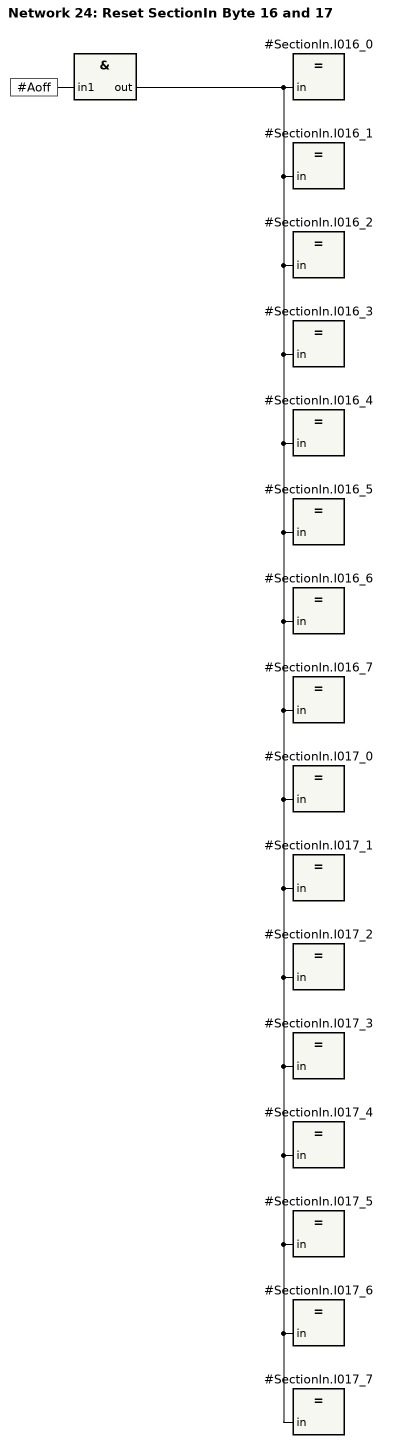
   #SectionIn.I016_0 := #Aoff;
   #SectionIn.I016_1 := #Aoff;
   #SectionIn.I016_2 := #Aoff;
   #SectionIn.I016_3 := #Aoff;
   #SectionIn.I016_4 := #Aoff;
   #SectionIn.I016_5 := #Aoff;
   #SectionIn.I016_6 := #Aoff;
   #SectionIn.I016_7 := #Aoff;
   #SectionIn.I017_0 := #Aoff;
   #SectionIn.I017_1 := #Aoff;
   #SectionIn.I017_2 := #Aoff;
   #SectionIn.I017_3 := #Aoff;
   #SectionIn.I017_4 := #Aoff;
   #SectionIn.I017_5 := #Aoff;
   #SectionIn.I017_6 := #Aoff;
   #SectionIn.I017_7 := #Aoff;
END_REGION

REGION Network 25: Reset SectionIn Byte 18 and 19
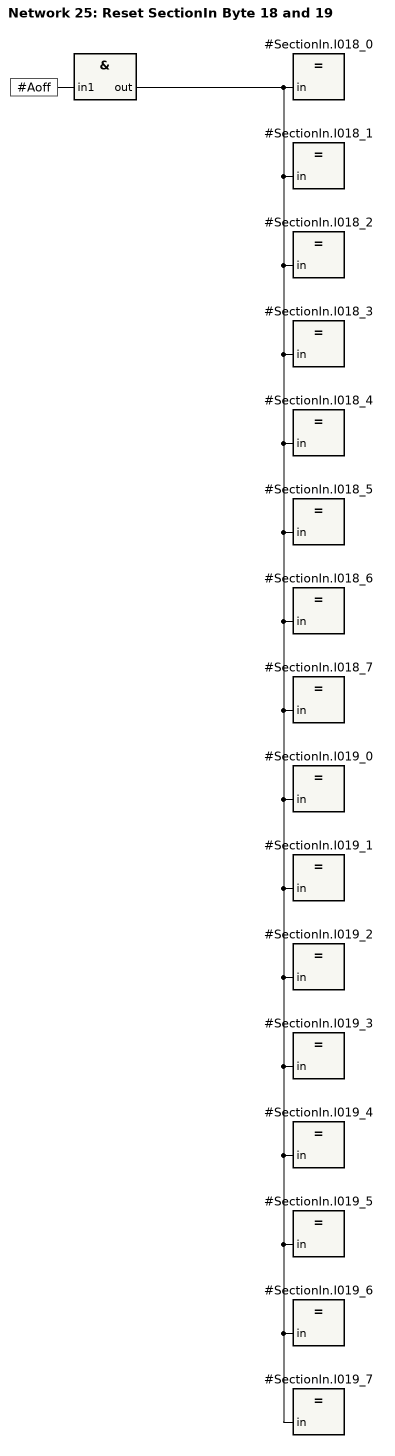
   #SectionIn.I018_0 := #Aoff;
   #SectionIn.I018_1 := #Aoff;
   #SectionIn.I018_2 := #Aoff;
   #SectionIn.I018_3 := #Aoff;
   #SectionIn.I018_4 := #Aoff;
   #SectionIn.I018_5 := #Aoff;
   #SectionIn.I018_6 := #Aoff;
   #SectionIn.I018_7 := #Aoff;
   #SectionIn.I019_0 := #Aoff;
   #SectionIn.I019_1 := #Aoff;
   #SectionIn.I019_2 := #Aoff;
   #SectionIn.I019_3 := #Aoff;
   #SectionIn.I019_4 := #Aoff;
   #SectionIn.I019_5 := #Aoff;
   #SectionIn.I019_6 := #Aoff;
   #SectionIn.I019_7 := #Aoff;
END_REGION

REGION Network 26: Reset SectionIn Byte 20 and 21
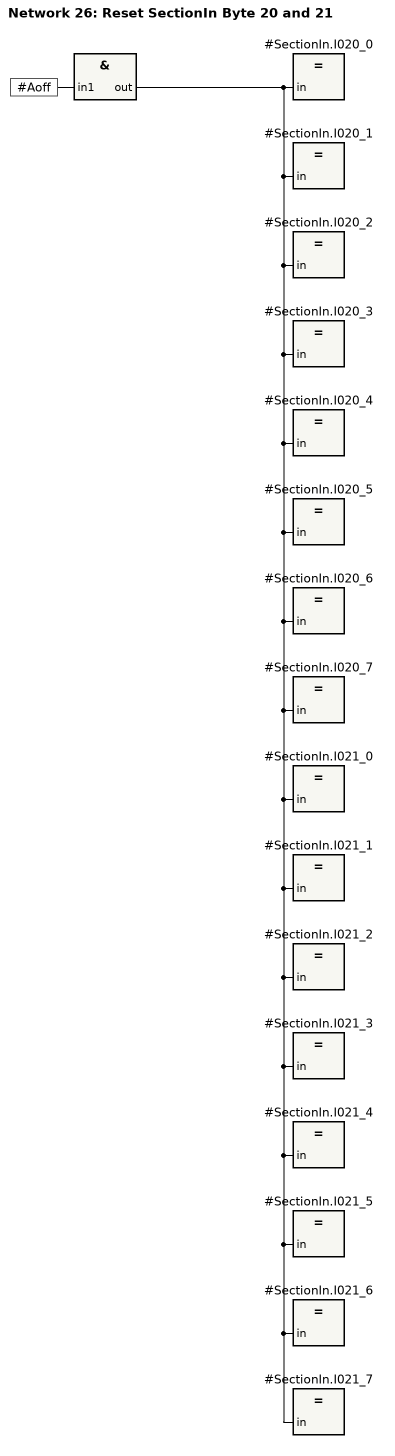
   #SectionIn.I020_0 := #Aoff;
   #SectionIn.I020_1 := #Aoff;
   #SectionIn.I020_2 := #Aoff;
   #SectionIn.I020_3 := #Aoff;
   #SectionIn.I020_4 := #Aoff;
   #SectionIn.I020_5 := #Aoff;
   #SectionIn.I020_6 := #Aoff;
   #SectionIn.I020_7 := #Aoff;
   #SectionIn.I021_0 := #Aoff;
   #SectionIn.I021_1 := #Aoff;
   #SectionIn.I021_2 := #Aoff;
   #SectionIn.I021_3 := #Aoff;
   #SectionIn.I021_4 := #Aoff;
   #SectionIn.I021_5 := #Aoff;
   #SectionIn.I021_6 := #Aoff;
   #SectionIn.I021_7 := #Aoff;
END_REGION

REGION Network 27: Reset SectionIn 22 to 99
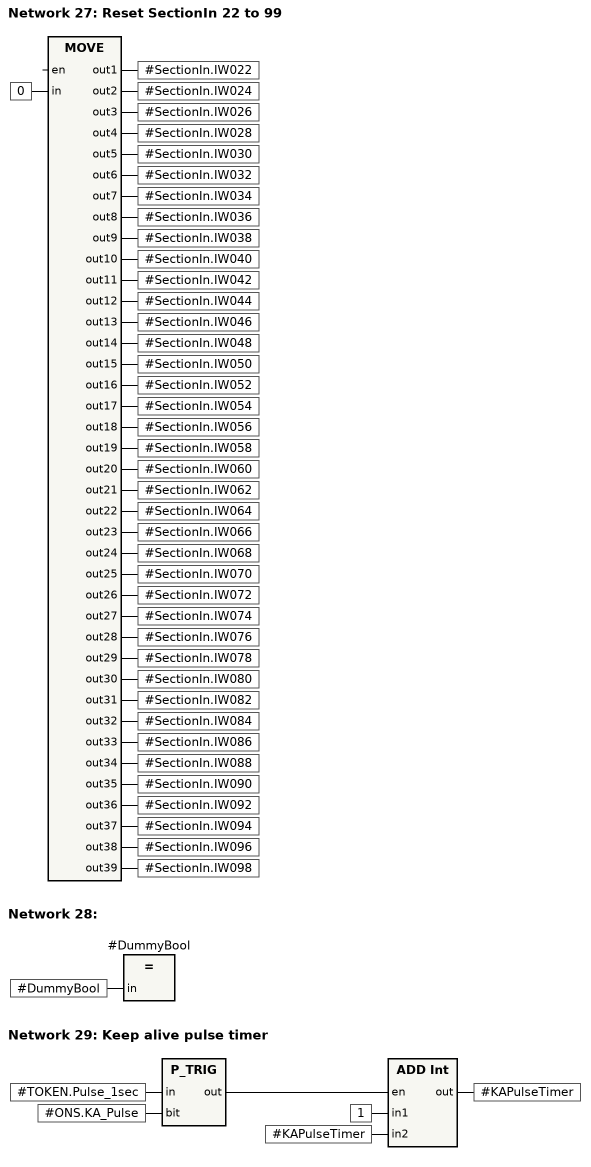
   #SectionIn.IW022 := 0;
   #SectionIn.IW024 := 0;
   #SectionIn.IW026 := 0;
   #SectionIn.IW028 := 0;
   #SectionIn.IW030 := 0;
   #SectionIn.IW032 := 0;
   #SectionIn.IW034 := 0;
   #SectionIn.IW036 := 0;
   #SectionIn.IW038 := 0;
   #SectionIn.IW040 := 0;
   #SectionIn.IW042 := 0;
   #SectionIn.IW044 := 0;
   #SectionIn.IW046 := 0;
   #SectionIn.IW048 := 0;
   #SectionIn.IW050 := 0;
   #SectionIn.IW052 := 0;
   #SectionIn.IW054 := 0;
   #SectionIn.IW056 := 0;
   #SectionIn.IW058 := 0;
   #SectionIn.IW060 := 0;
   #SectionIn.IW062 := 0;
   #SectionIn.IW064 := 0;
   #SectionIn.IW066 := 0;
   #SectionIn.IW068 := 0;
   #SectionIn.IW070 := 0;
   #SectionIn.IW072 := 0;
   #SectionIn.IW074 := 0;
   #SectionIn.IW076 := 0;
   #SectionIn.IW078 := 0;
   #SectionIn.IW080 := 0;
   #SectionIn.IW082 := 0;
   #SectionIn.IW084 := 0;
   #SectionIn.IW086 := 0;
   #SectionIn.IW088 := 0;
   #SectionIn.IW090 := 0;
   #SectionIn.IW092 := 0;
   #SectionIn.IW094 := 0;
   #SectionIn.IW096 := 0;
   #SectionIn.IW098 := 0;
END_REGION

REGION Network 28
   Res1:
   #DummyBool := #DummyBool;
END_REGION

REGION Network 29: Keep alive pulse timer
   #_w1 := #TOKEN.Pulse_1sec AND NOT #ONS.KA_Pulse;   // rising edge
   #ONS.KA_Pulse := #TOKEN.Pulse_1sec;
   IF #_w1 THEN #KAPulseTimer := 1 + #KAPulseTimer; END_IF;
END_REGION

REGION Network 30: Keep alive pulse generated
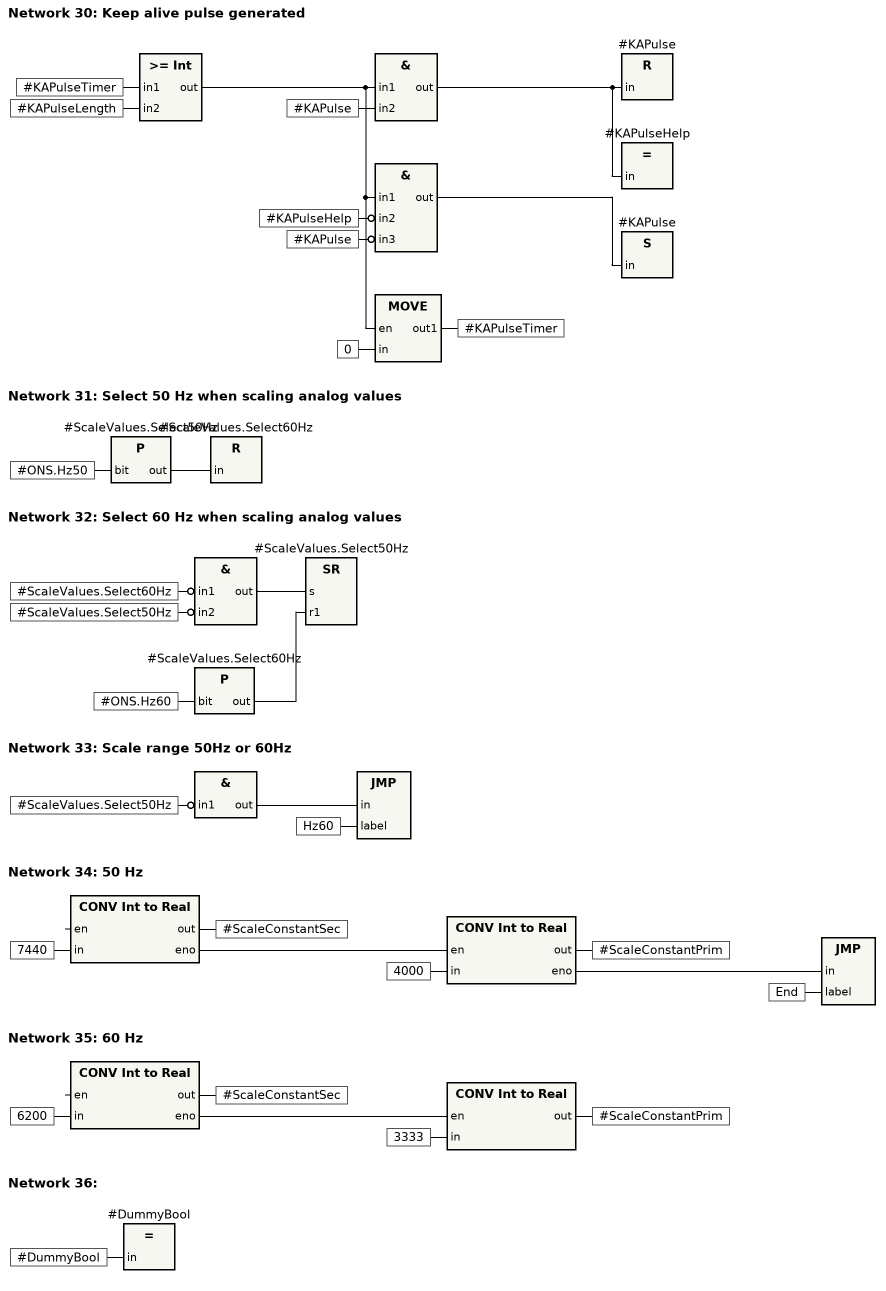
   #_w1 := #KAPulseTimer >= #KAPulseLength;
   #_w2 := #_w1 AND #KAPulse;
   IF #_w2 THEN #KAPulse := FALSE; END_IF;
   #KAPulseHelp := #_w2;
   IF #_w1 AND NOT #KAPulseHelp AND NOT #KAPulse THEN #KAPulse := TRUE; END_IF;
   IF #_w1 THEN #KAPulseTimer := 0; END_IF;
END_REGION

REGION Network 31: Select 50 Hz when scaling analog values
   #_w1 := #ScaleValues.Select50Hz AND NOT #ONS.Hz50;   // rising edge of #ScaleValues.Select50Hz
   #ONS.Hz50 := #ScaleValues.Select50Hz;
   IF #_w1 THEN #ScaleValues.Select60Hz := FALSE; END_IF;
END_REGION

REGION Network 32: Select 60 Hz when scaling analog values
   #_w1 := #ScaleValues.Select60Hz AND NOT #ONS.Hz60;   // rising edge of #ScaleValues.Select60Hz
   #ONS.Hz60 := #ScaleValues.Select60Hz;
   IF NOT #ScaleValues.Select60Hz AND NOT #ScaleValues.Select50Hz THEN
       #ScaleValues.Select50Hz := TRUE;   // SR flip-flop
   END_IF;
   IF #_w1 THEN #ScaleValues.Select50Hz := FALSE; END_IF;
END_REGION

REGION Network 33: Scale range 50Hz or 60Hz
   // Jump if not 50Hz
   IF NOT #ScaleValues.Select50Hz THEN GOTO Hz60; END_IF;
END_REGION

REGION Network 34: 50 Hz
   #ScaleConstantSec := INT_TO_REAL(7440);
   #ScaleConstantPrim := INT_TO_REAL(4000);
   GOTO End;
END_REGION

REGION Network 35: 60 Hz
   Hz60:
   #ScaleConstantSec := INT_TO_REAL(6200);
   #ScaleConstantPrim := INT_TO_REAL(3333);
END_REGION

REGION Network 36
   End:
   #DummyBool := #DummyBool;
END_REGION

REGION Network 37: Latch Acknowledge signal from ECS section
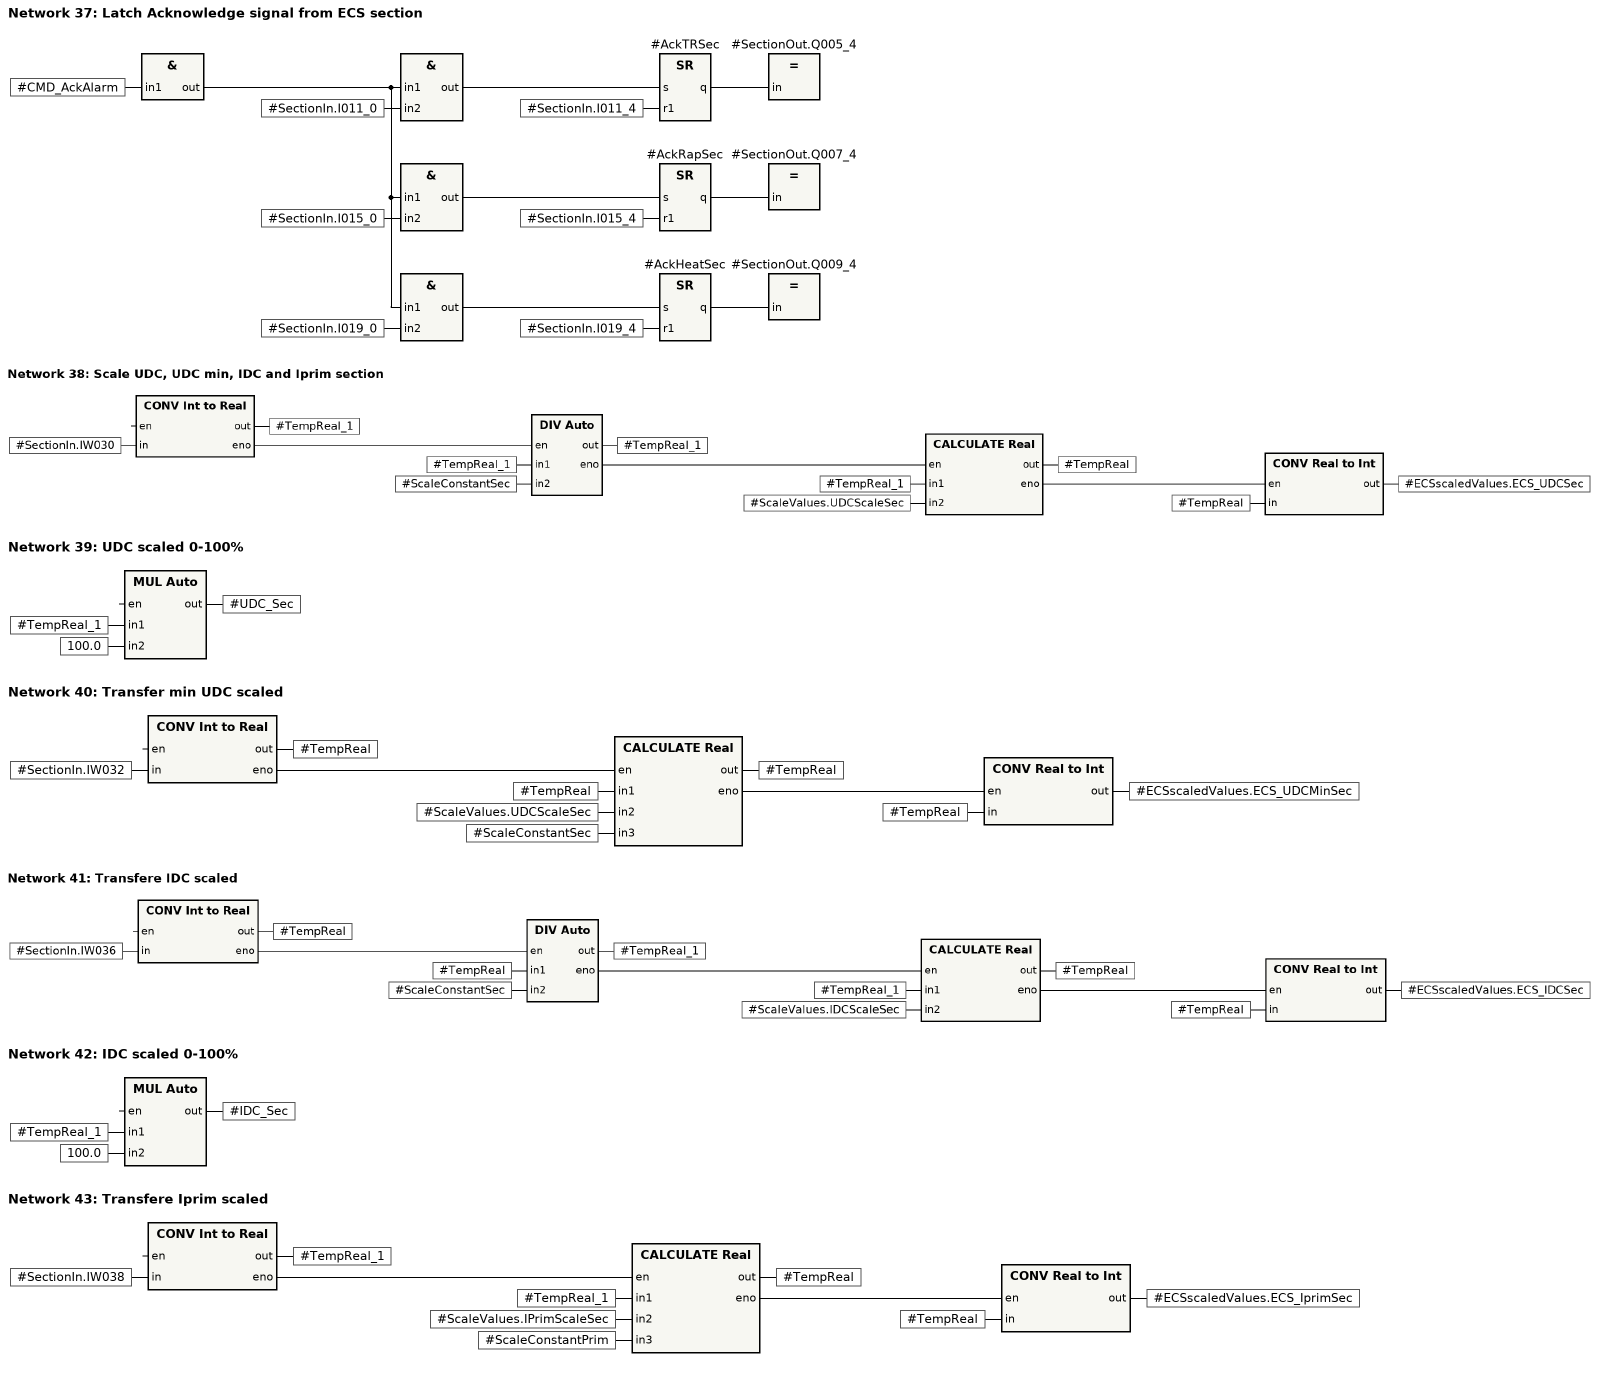
   IF #CMD_AckAlarm AND #SectionIn.I011_0 THEN
       #AckTRSec := TRUE;   // SR flip-flop
   END_IF;
   IF #SectionIn.I011_4 THEN #AckTRSec := FALSE; END_IF;
   #SectionOut.Q005_4 := #AckTRSec;
   IF #CMD_AckAlarm AND #SectionIn.I015_0 THEN
       #AckRapSec := TRUE;   // SR flip-flop
   END_IF;
   IF #SectionIn.I015_4 THEN #AckRapSec := FALSE; END_IF;
   #SectionOut.Q007_4 := #AckRapSec;
   IF #CMD_AckAlarm AND #SectionIn.I019_0 THEN
       #AckHeatSec := TRUE;   // SR flip-flop
   END_IF;
   IF #SectionIn.I019_4 THEN #AckHeatSec := FALSE; END_IF;
   #SectionOut.Q009_4 := #AckHeatSec;
END_REGION

REGION Network 38: Scale UDC, UDC min, IDC and Iprim section
   // Transfer UDC scaled
   // Build 002 : 26 March 2019 - ECS_UDCSec/ECS_UDCMinSec were mul by 10.0 before and the same is removed
   #TempReal_1 := INT_TO_REAL(#SectionIn.IW030);
   #TempReal_1 := #TempReal_1 / #ScaleConstantSec;
   #TempReal := ROUND(#TempReal_1*#ScaleValues.UDCScaleSec);
   #ECSscaledValues.ECS_UDCSec := REAL_TO_INT(#TempReal);
END_REGION

REGION Network 39: UDC scaled 0-100%
   #UDC_Sec := #TempReal_1 * 100.0;
END_REGION

REGION Network 40: Transfer min UDC scaled
   // Build 002 : 26 March 2019 - ECS_UDCSec/ECS_UDCMinSec were mul by 10.0 before and the same is removed
   #TempReal := INT_TO_REAL(#SectionIn.IW032);
   #TempReal := ROUND((#TempReal*#ScaleValues.UDCScaleSec)/#ScaleConstantSec);
   #ECSscaledValues.ECS_UDCMinSec := REAL_TO_INT(#TempReal);
END_REGION

REGION Network 41: Transfere IDC scaled
   #TempReal := INT_TO_REAL(#SectionIn.IW036);
   #TempReal_1 := #TempReal / #ScaleConstantSec;
   #TempReal := ROUND(#TempReal_1*#ScaleValues.IDCScaleSec);
   #ECSscaledValues.ECS_IDCSec := REAL_TO_INT(#TempReal);
END_REGION

REGION Network 42: IDC scaled 0-100%
   #IDC_Sec := #TempReal_1 * 100.0;
END_REGION

REGION Network 43: Transfere Iprim scaled
   #TempReal_1 := INT_TO_REAL(#SectionIn.IW038);
   #TempReal := ROUND((#TempReal_1*#ScaleValues.IPrimScaleSec)/#ScaleConstantPrim);
   #ECSscaledValues.ECS_IprimSec := REAL_TO_INT(#TempReal);
END_REGION

REGION Network 44: Transfer general outputs to gateway
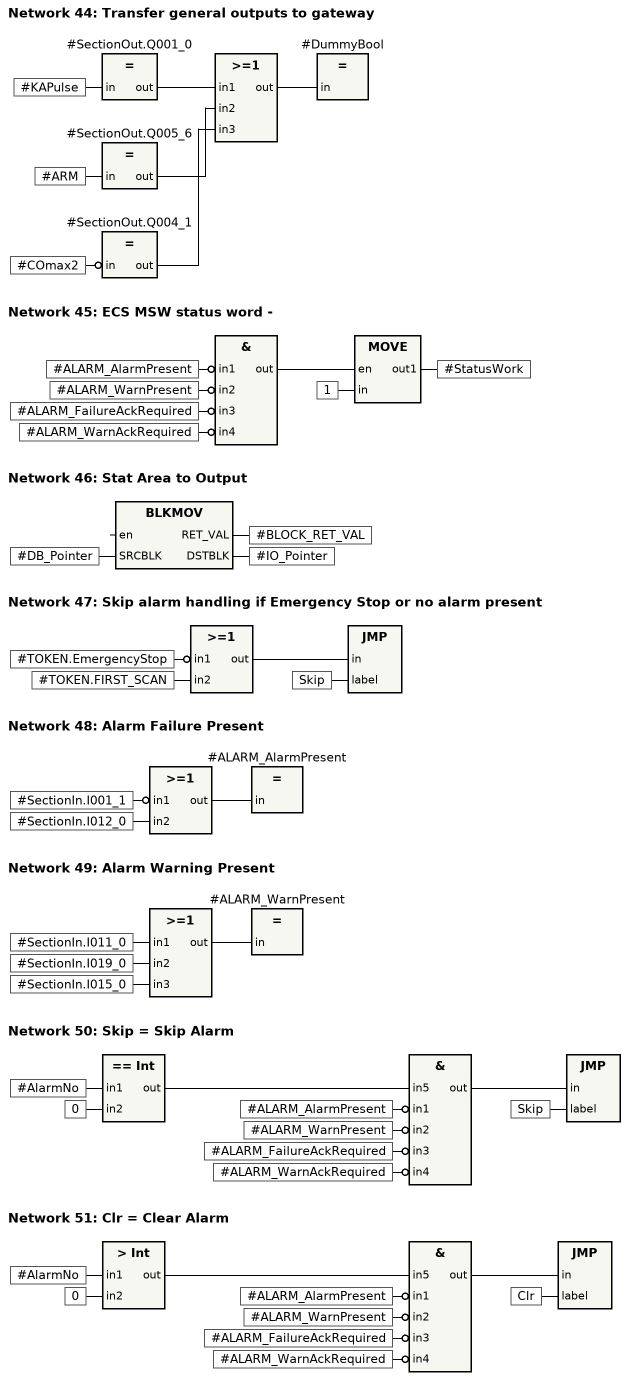
   #SectionOut.Q001_0 := #KAPulse;
   #SectionOut.Q005_6 := #ARM;
   #SectionOut.Q004_1 := NOT #COmax2;
   #DummyBool := #KAPulse OR #ARM OR NOT #COmax2;
END_REGION

REGION Network 45: ECS MSW status word -
   IF NOT #ALARM_AlarmPresent AND NOT #ALARM_WarnPresent AND NOT #ALARM_FailureAckRequired AND NOT #ALARM_WarnAckRequired THEN
       #StatusWork := 1;
   END_IF;
END_REGION

REGION Network 46: Stat Area to Output
   #BLOCK_RET_VAL := BLKMOV(SRCBLK := #DB_Pointer, DSTBLK => #IO_Pointer);
END_REGION

REGION Network 47: Skip alarm handling if Emergency Stop or no alarm present
   // Skip = Skip Alarm
   IF NOT #TOKEN.EmergencyStop OR #TOKEN.FIRST_SCAN THEN GOTO Skip; END_IF;
END_REGION

REGION Network 48: Alarm Failure Present
   #ALARM_AlarmPresent := NOT #SectionIn.I001_1 OR #SectionIn.I012_0;
END_REGION

REGION Network 49: Alarm Warning Present
   #ALARM_WarnPresent := #SectionIn.I011_0 OR #SectionIn.I019_0 OR #SectionIn.I015_0;
END_REGION

REGION Network 50: Skip = Skip Alarm
   IF (#AlarmNo = 0) AND NOT #ALARM_AlarmPresent AND NOT #ALARM_WarnPresent AND NOT #ALARM_FailureAckRequired AND NOT #ALARM_WarnAckRequired THEN
       GOTO Skip;
   END_IF;
END_REGION

REGION Network 51: Clr = Clear Alarm
   IF (#AlarmNo > 0) AND NOT #ALARM_AlarmPresent AND NOT #ALARM_WarnPresent AND NOT #ALARM_FailureAckRequired AND NOT #ALARM_WarnAckRequired THEN
       GOTO Clr;
   END_IF;
END_REGION

REGION Network 52: Ack = Alarm Acknowledge
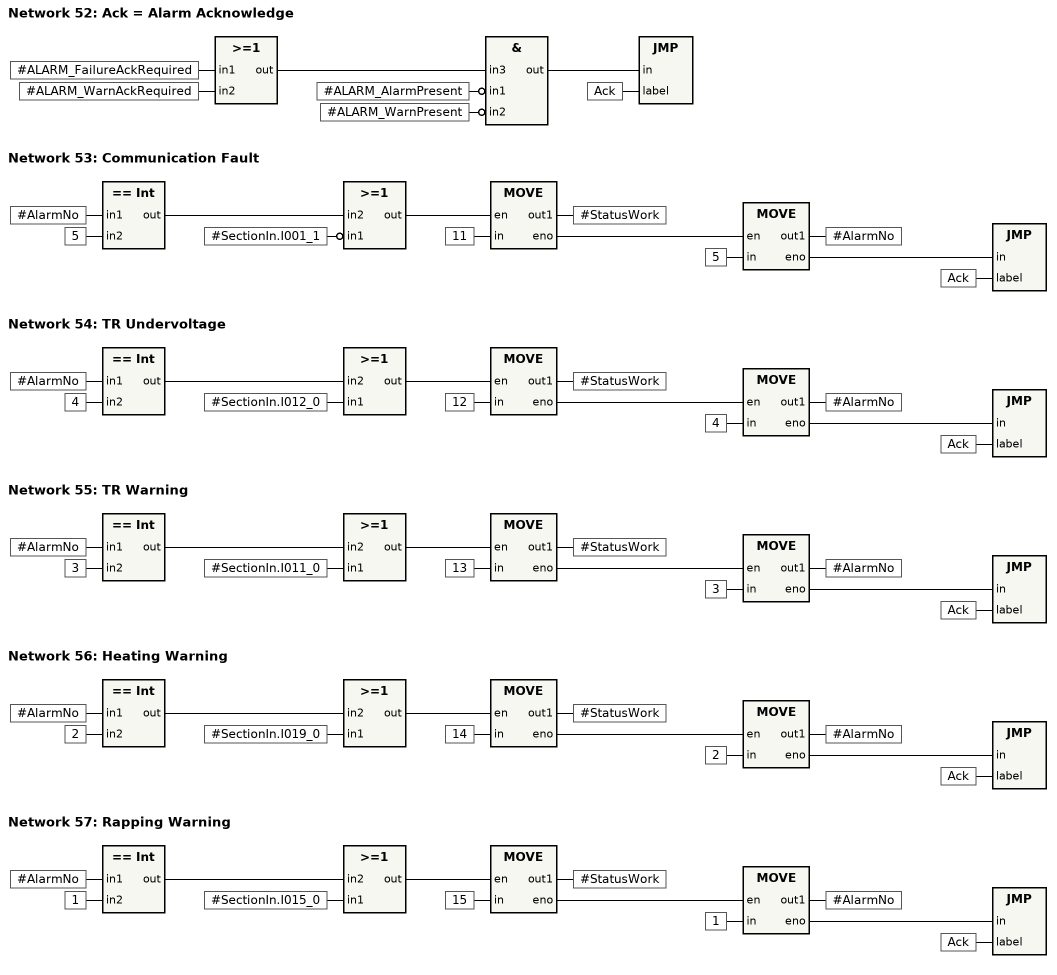
   IF (#ALARM_FailureAckRequired OR #ALARM_WarnAckRequired) AND NOT #ALARM_AlarmPresent AND NOT #ALARM_WarnPresent THEN
       GOTO Ack;
   END_IF;
END_REGION

REGION Network 53: Communication Fault
   // ENO of a box is taken as its EN; it also drops when the box reports an error
   #_w1 := (#AlarmNo = 5) OR NOT #SectionIn.I001_1;
   IF #_w1 THEN
       #StatusWork := 11;
       #AlarmNo := 5;
       GOTO Ack;
   END_IF;
END_REGION

REGION Network 54: TR Undervoltage
   // ENO of a box is taken as its EN; it also drops when the box reports an error
   #_w1 := (#AlarmNo = 4) OR #SectionIn.I012_0;
   IF #_w1 THEN
       #StatusWork := 12;
       #AlarmNo := 4;
       GOTO Ack;
   END_IF;
END_REGION

REGION Network 55: TR Warning
   // ENO of a box is taken as its EN; it also drops when the box reports an error
   #_w1 := (#AlarmNo = 3) OR #SectionIn.I011_0;
   IF #_w1 THEN
       #StatusWork := 13;
       #AlarmNo := 3;
       GOTO Ack;
   END_IF;
END_REGION

REGION Network 56: Heating Warning
   // ENO of a box is taken as its EN; it also drops when the box reports an error
   #_w1 := (#AlarmNo = 2) OR #SectionIn.I019_0;
   IF #_w1 THEN
       #StatusWork := 14;
       #AlarmNo := 2;
       GOTO Ack;
   END_IF;
END_REGION

REGION Network 57: Rapping Warning
   // ENO of a box is taken as its EN; it also drops when the box reports an error
   #_w1 := (#AlarmNo = 1) OR #SectionIn.I015_0;
   IF #_w1 THEN
       #StatusWork := 15;
       #AlarmNo := 1;
       GOTO Ack;
   END_IF;
END_REGION

REGION Network 58: Alarm Acknowledge
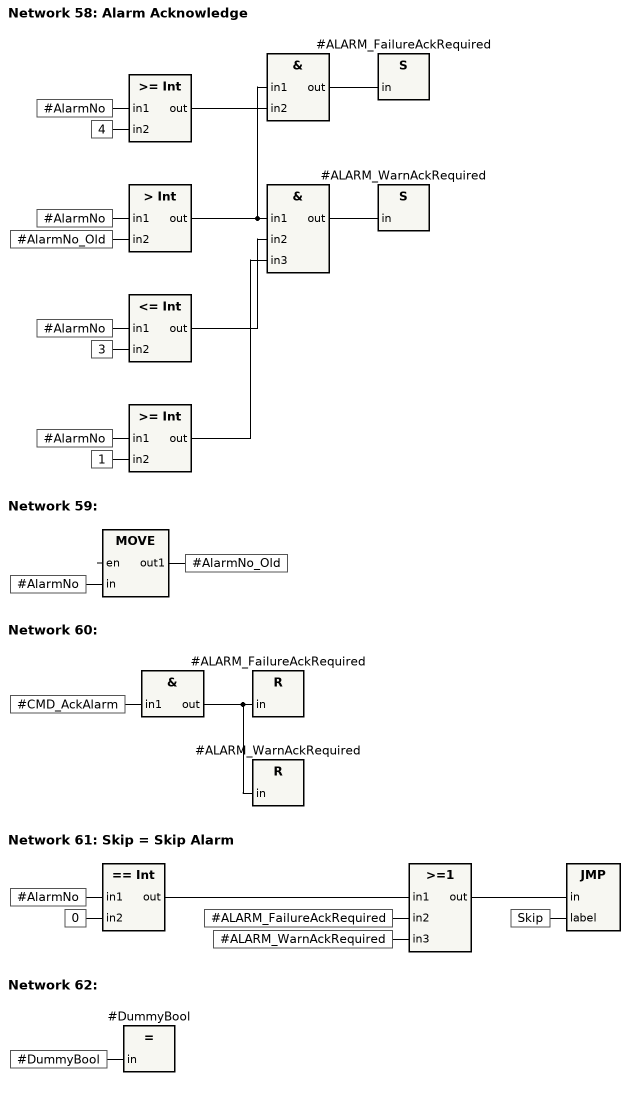
   Ack:
   #_w1 := #AlarmNo > #AlarmNo_Old;
   IF #_w1 AND (#AlarmNo >= 4) THEN #ALARM_FailureAckRequired := TRUE; END_IF;
   IF #_w1 AND (#AlarmNo <= 3) AND (#AlarmNo >= 1) THEN #ALARM_WarnAckRequired := TRUE; END_IF;
END_REGION

REGION Network 59
   #AlarmNo_Old := #AlarmNo;
END_REGION

REGION Network 60
   IF #CMD_AckAlarm THEN
       #ALARM_FailureAckRequired := FALSE;
       #ALARM_WarnAckRequired := FALSE;
   END_IF;
END_REGION

REGION Network 61: Skip = Skip Alarm
   IF (#AlarmNo = 0) OR #ALARM_FailureAckRequired OR #ALARM_WarnAckRequired THEN GOTO Skip; END_IF;
END_REGION

REGION Network 62
   Clr:
   #DummyBool := #DummyBool;
END_REGION

REGION Network 63
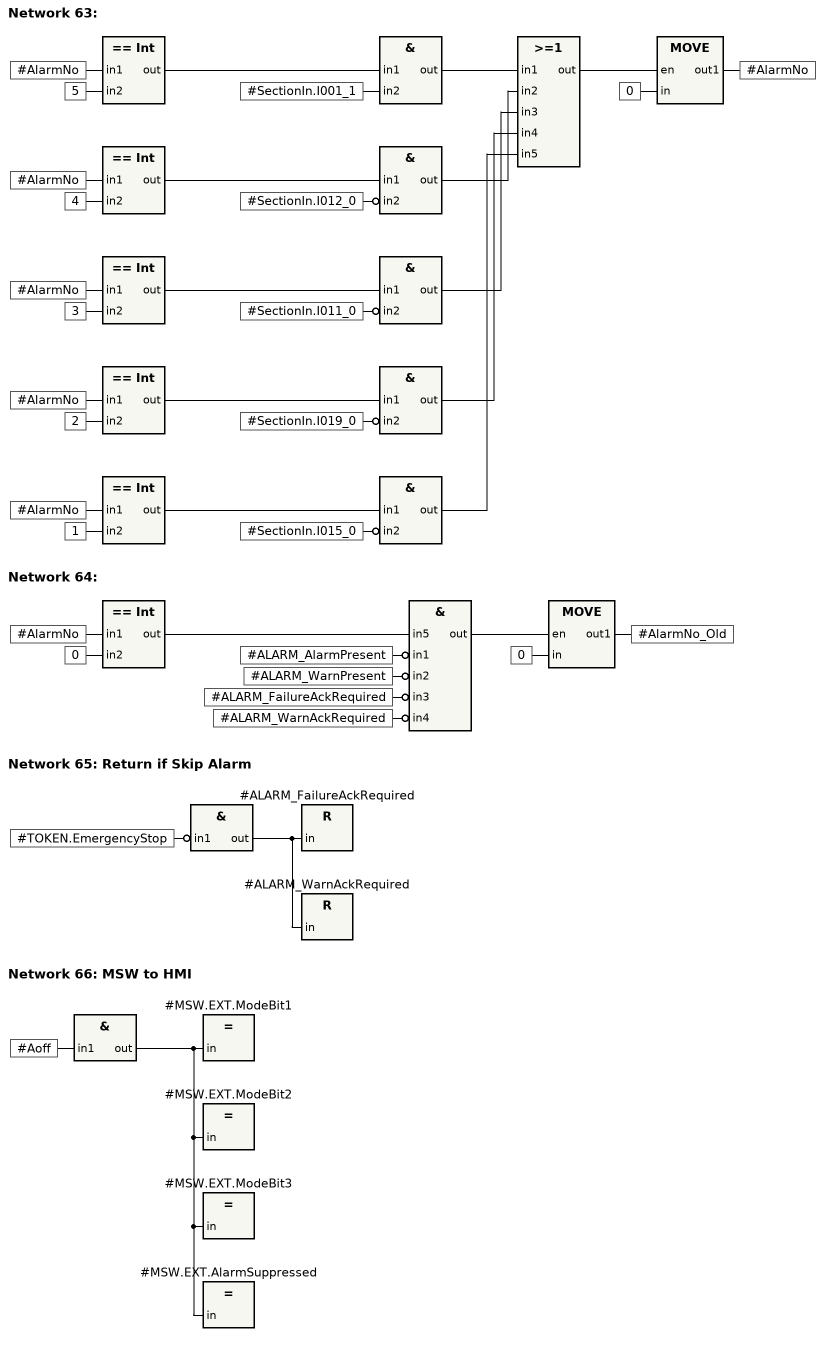
   IF ((#AlarmNo = 5) AND #SectionIn.I001_1) OR ((#AlarmNo = 4) AND NOT #SectionIn.I012_0) OR ((#AlarmNo = 3) AND NOT #SectionIn.I011_0) OR ((#AlarmNo = 2) AND NOT #SectionIn.I019_0) OR ((#AlarmNo = 1) AND NOT #SectionIn.I015_0) THEN
       #AlarmNo := 0;
   END_IF;
END_REGION

REGION Network 64
   IF (#AlarmNo = 0) AND NOT #ALARM_AlarmPresent AND NOT #ALARM_WarnPresent AND NOT #ALARM_FailureAckRequired AND NOT #ALARM_WarnAckRequired THEN
       #AlarmNo_Old := 0;
   END_IF;
END_REGION

REGION Network 65: Return if Skip Alarm
   Skip:
   IF NOT #TOKEN.EmergencyStop THEN
       #ALARM_FailureAckRequired := FALSE;
       #ALARM_WarnAckRequired := FALSE;
   END_IF;
END_REGION

REGION Network 66: MSW to HMI
   #MSW.EXT.ModeBit1 := #Aoff;
   #MSW.EXT.ModeBit2 := #Aoff;
   #MSW.EXT.ModeBit3 := #Aoff;
   #MSW.EXT.AlarmSuppressed := #Aoff;
END_REGION

REGION Network 67
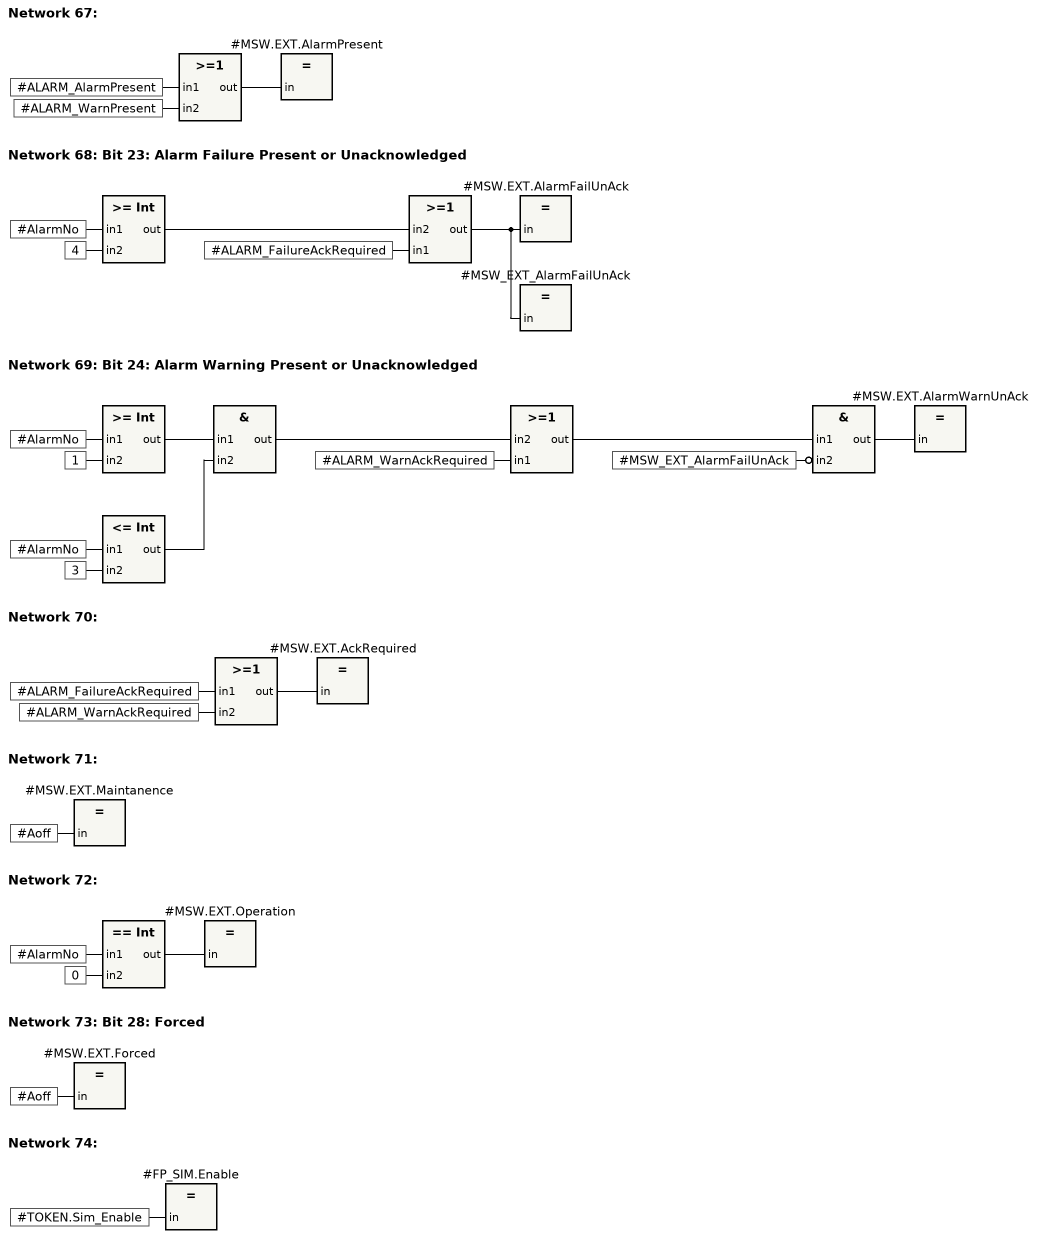
   #MSW.EXT.AlarmPresent := #ALARM_AlarmPresent OR #ALARM_WarnPresent;
END_REGION

REGION Network 68: Bit 23: Alarm Failure Present or Unacknowledged
   #MSW.EXT.AlarmFailUnAck := (#AlarmNo >= 4) OR #ALARM_FailureAckRequired;
   #MSW_EXT_AlarmFailUnAck := #MSW.EXT.AlarmFailUnAck;
END_REGION

REGION Network 69: Bit 24: Alarm Warning Present or Unacknowledged
   #MSW.EXT.AlarmWarnUnAck := (((#AlarmNo >= 1) AND (#AlarmNo <= 3)) OR #ALARM_WarnAckRequired) AND NOT #MSW_EXT_AlarmFailUnAck;
END_REGION

REGION Network 70
   #MSW.EXT.AckRequired := #ALARM_FailureAckRequired OR #ALARM_WarnAckRequired;
END_REGION

REGION Network 71
   #MSW.EXT.Maintanence := #Aoff;
END_REGION

REGION Network 72
   #MSW.EXT.Operation := #AlarmNo = 0;
END_REGION

REGION Network 73: Bit 28: Forced
   #MSW.EXT.Forced := #Aoff;
END_REGION

REGION Network 74
   #FP_SIM.Enable := #TOKEN.Sim_Enable;
END_REGION

REGION Network 75: MSW & TIMESTAMP TO HMI
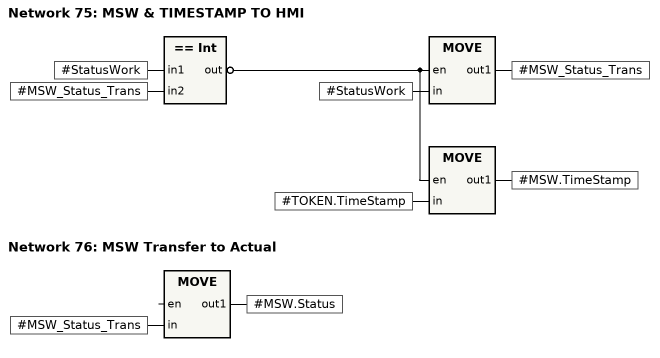
   #_w1 := NOT (#StatusWork = #MSW_Status_Trans);
   IF #_w1 THEN
       #MSW_Status_Trans := #StatusWork;
       #MSW.TimeStamp := #TOKEN.TimeStamp;
   END_IF;
END_REGION

REGION Network 76: MSW Transfer to Actual
   #MSW.Status := #MSW_Status_Trans;
END_REGION
END_FUNCTION_BLOCK

FUNCTION_BLOCK "ACESYS_SEL_ANALOG"   // FB234, FBD
TITLE = ACESYS V8.0 - Build 002 - Select Analog Block
{ S7_Optimized_Access := 'FALSE' }
AUTHOR : FLSmidth
FAMILY : ACESYS
NAME : SEL_ALOG
VERSION : 8.0
   VAR_INPUT
      X1 : Real;   // Signal 1
      X2 : Real;   // Signal 2
      X3 : Real;   // Signal 3
      X1_OK : Bool;   // Signal 1 Enable
      X2_OK : Bool;   // Signal 2 Enable
      X3_OK : Bool;   // Signal 3 Enable
   END_VAR
   VAR_OUTPUT
      SEL_X1 : Bool;   // Signal 1 Selected
      SEL_X2 : Bool;   // Signal 2 Selected
      SEL_X3 : Bool;   // Signal 3 Selected
      AL_X1 : Bool;   // Alarm Signal 1 (1 = OK)
      AL_X2 : Bool;   // Alarm Signal 2 (1 = OK)
      AL_X3 : Bool;   // Alarm Signal 3 (1 = OK)
      AVG : Real;   // Average
      MSW : "ACESYS_HMI_STAT_ANALOG";
   END_VAR
   VAR_IN_OUT
      TOKEN : "ACESYS_TOKEN";
   END_VAR
   VAR
      BlockInfo : Struct
         Ace_Version : Int;   // Acesys Block Version Number
         Ace_BuildNo : Int;   // Acesys Block Build Number
         DB_Number : Int;   // Block Instance DB Number
      END_STRUCT;
      FP_CMD : Struct   // Faceplate Commands
         Spare_08 : Bool;
         Spare_09 : Bool;
         Spare_10 : Bool;
         Spare_11 : Bool;
         Spare_12 : Bool;
         Spare_13 : Bool;
         Spare_14 : Bool;
         AckAlarm : Bool;
         Spare_00 : Bool;
         Spare_01 : Bool;
         Spare_02 : Bool;
         Spare_03 : Bool;
         Spare_04 : Bool;
         Spare_05 : Bool;
         Spare_06 : Bool;
         Spare_07 : Bool;
      END_STRUCT;
      FP_SEL : Struct   // Faceplate Selection
         X1 : Bool := TRUE;   // Select X1 from Faceplate
         X2 : Bool := TRUE;   // Select X2 from Faceplate
         X3 : Bool := TRUE;   // Select X3 from Faceplate
         Type2 : Bool;   // Select 2 Sensors
         Type3 : Bool;   // Select 3 Sensors
         MaxVal : Bool;   // Select Max Value (2 sensors)
         MinVal : Bool;   // Select Min Value (2 sensors)
         Spare9 : Bool;
         Spare8 : Bool;
         Spare7 : Bool;
         Spare6 : Bool;
         Spare5 : Bool;
         Spare4 : Bool;
         Spare3 : Bool;
         Spare2 : Bool;
         Spare1 : Bool;
      END_STRUCT;
      FP_SHOW : Struct   // Faceplate Show Object
         X1 : Bool;   // Show X1 on Faceplate
         X2 : Bool;   // Show X2 on Faceplate
         X3 : Bool;   // Show X3 on Faceplate
      END_STRUCT;
      FP_PARM : Struct   // Faceplate Parameters
         MaxDiff : Real := 10.0;   // Max Diff SP
         AL_Delay_Pre : Int := 3;   // Alarm Delay Pre
         AL_Delay_Acc : Int;   // Alarm Delay ACC
      END_STRUCT;
      ONS : Struct
         SecPulse1 : Bool;   // Oneshot Bit
         SecPulse2 : Bool;   // Oneshot Bit
         Sel_Type2 : Bool;   // Oneshot Bit
         Sel_Type3 : Bool;   // Oneshot Bit
         Sel_High : Bool;   // Oneshot Bit
         Sel_Low : Bool;   // Oneshot Bit
         Sel_Max : Bool;   // Oneshot Bit
         Sel_Min : Bool;   // Oneshot Bit
         Acknowledge : Bool;
         Spare7 : Bool;
         Spare6 : Bool;
         Spare5 : Bool;
         Spare4 : Bool;
         Spare3 : Bool;
         Spare2 : Bool;
         Spare1 : Bool;
      END_STRUCT;
      Sec_Pulse : Bool;   // Pulse Every Second
      Sig1_3_NotOK : Bool;
      Sig1_2_NotOK : Bool;
      Sig2_3_NotOK : Bool;
      Sig1_Deviation : Bool;   // Signal 1 Deviation
      Sig2_Deviation : Bool;   // Signal 2 Deviation
      Sig3_Deviation : Bool;   // Signal 3 Deviation
      CMD_Acknowledge : Bool;   // Internal Acknowledge
      ALARM_SuppresionActiv : Bool;   // Internal Alarm Supression
      ALARM_AlarmPresent : Bool;
      ALARM_Failure_Ack_Requ : Bool;
      ALARM_Warn_Ack_Requ : Bool;
      ALARM_WarnPresent : Bool;
      SEL_X1_int : Bool;   // Signal 1 Selected
      SEL_X2_int : Bool;   // Signal 2 Selected
      SEL_X3_int : Bool;   // Signal 3 Selected
      Sig1_Fault : Bool;   // Signal 1 Fault
      Sig2_Fault : Bool;   // Signal 2 Fault
      Sig3_Fault : Bool;   // Signal 3 Fault
      Sig1_3_TimerMEM : Int;   // Timer Memory Register
      Sig1_2_TimerMEM : Int;   // Timer Memory Register
      Sig2_3_TimerMEM : Int;   // Timer Memory Register
      AlarmNo : Int;   // Alarm Number
      AlarmNo_Old : Int;   // Old Alarm Number
      StatusWork : Int;   // Internal ECS Status
      No_X : Real;   // Number of Signals in Calculation
      Sum_X : Real;   // Total Signal Value of X:s
      MinMaxVal : Real;   // Selected Min Max Val (for Type-2)
      OUT : Struct
         SEL_X1 : Bool;
         SEL_X2 : Bool;
         SEL_X3 : Bool;
         AL_X1 : Bool;
         AL_X2 : Bool;
         AL_X3 : Bool;
         AVG : Real;
         MSW_EXT_ALARMFAILUNACK : Bool;
      END_STRUCT;
      MSW_Status_Trans : Int;
   END_VAR
   VAR_TEMP
      AOn : Bool;   // Always On
      AOff : Bool;   // Always Off
      DummyBool : Bool;
      DummyReal_1 : Real;
      DummyReal_2 : Real;
   END_VAR
   VAR_TEMP   // added for the SCL form of the ladder/FBD networks
      _w1 : Bool;
      _w2 : Bool;
   END_VAR
BEGIN

REGION Network 1: Always On
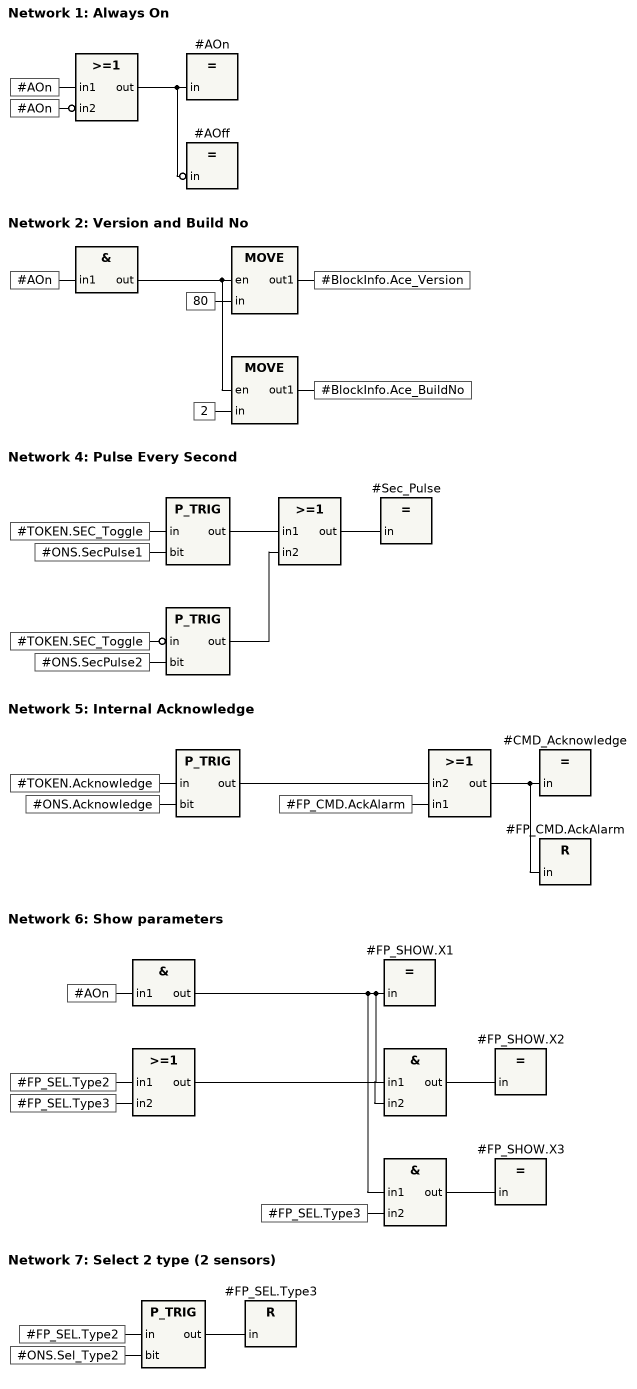
   #AOn := #AOn OR NOT #AOn;
   #AOff := NOT #AOn;
END_REGION

REGION Network 2: Version and Build No
   IF #AOn THEN
       #BlockInfo.Ace_Version := 80;
       #BlockInfo.Ace_BuildNo := 2;
   END_IF;
END_REGION

REGION Network 3 (STL): Instance DB Number to Faceplate
         L     DINO;
         T     #BlockInfo.DB_Number;
END_REGION

REGION Network 4: Pulse Every Second
   #_w1 := #TOKEN.SEC_Toggle AND NOT #ONS.SecPulse1;   // rising edge
   #ONS.SecPulse1 := #TOKEN.SEC_Toggle;
   #_w2 := NOT #TOKEN.SEC_Toggle AND NOT #ONS.SecPulse2;   // rising edge
   #ONS.SecPulse2 := NOT #TOKEN.SEC_Toggle;
   #Sec_Pulse := #_w1 OR #_w2;
END_REGION

REGION Network 5: Internal Acknowledge
   #_w1 := #TOKEN.Acknowledge AND NOT #ONS.Acknowledge;   // rising edge
   #ONS.Acknowledge := #TOKEN.Acknowledge;
   #CMD_Acknowledge := #_w1 OR #FP_CMD.AckAlarm;
   IF #CMD_Acknowledge THEN #FP_CMD.AckAlarm := FALSE; END_IF;
END_REGION

REGION Network 6: Show parameters
   #FP_SHOW.X1 := #AOn;
   #FP_SHOW.X2 := #AOn AND (#FP_SEL.Type2 OR #FP_SEL.Type3);
   #FP_SHOW.X3 := #AOn AND #FP_SEL.Type3;
END_REGION

REGION Network 7: Select 2 type (2 sensors)
   #_w1 := #FP_SEL.Type2 AND NOT #ONS.Sel_Type2;   // rising edge
   #ONS.Sel_Type2 := #FP_SEL.Type2;
   IF #_w1 THEN #FP_SEL.Type3 := FALSE; END_IF;
END_REGION

REGION Network 8: Select 3 type (3 sensors)
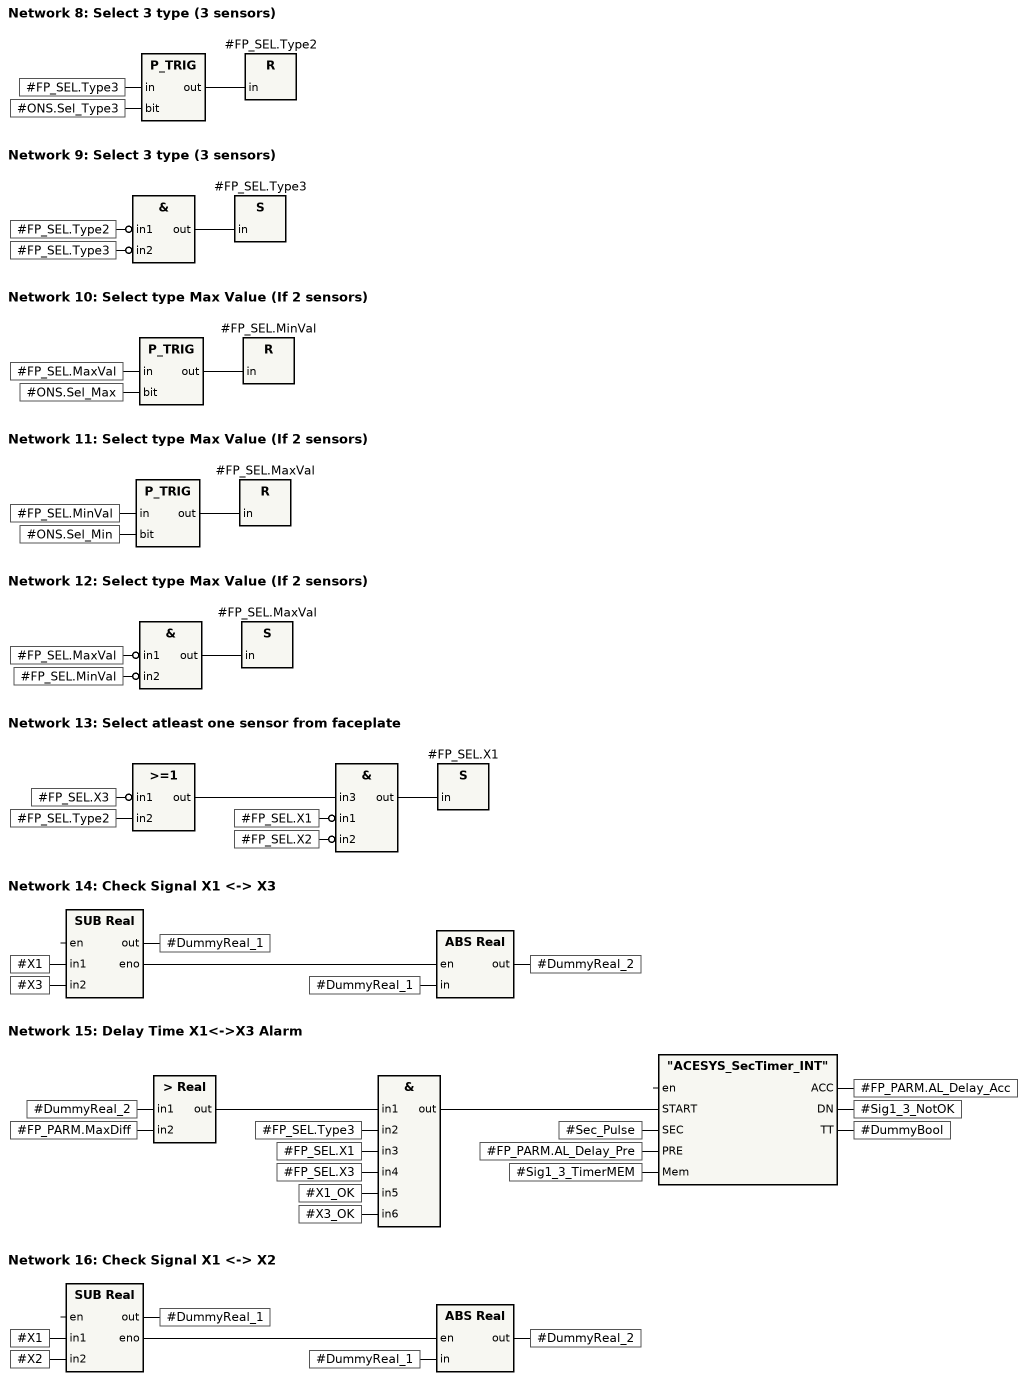
   #_w1 := #FP_SEL.Type3 AND NOT #ONS.Sel_Type3;   // rising edge
   #ONS.Sel_Type3 := #FP_SEL.Type3;
   IF #_w1 THEN #FP_SEL.Type2 := FALSE; END_IF;
END_REGION

REGION Network 9: Select 3 type (3 sensors)
   IF NOT #FP_SEL.Type2 AND NOT #FP_SEL.Type3 THEN #FP_SEL.Type3 := TRUE; END_IF;
END_REGION

REGION Network 10: Select type Max Value (If 2 sensors)
   #_w1 := #FP_SEL.MaxVal AND NOT #ONS.Sel_Max;   // rising edge
   #ONS.Sel_Max := #FP_SEL.MaxVal;
   IF #_w1 THEN #FP_SEL.MinVal := FALSE; END_IF;
END_REGION

REGION Network 11: Select type Max Value (If 2 sensors)
   #_w1 := #FP_SEL.MinVal AND NOT #ONS.Sel_Min;   // rising edge
   #ONS.Sel_Min := #FP_SEL.MinVal;
   IF #_w1 THEN #FP_SEL.MaxVal := FALSE; END_IF;
END_REGION

REGION Network 12: Select type Max Value (If 2 sensors)
   IF NOT #FP_SEL.MaxVal AND NOT #FP_SEL.MinVal THEN #FP_SEL.MaxVal := TRUE; END_IF;
END_REGION

REGION Network 13: Select atleast one sensor from faceplate
   // Build 002 - 17. Jun 2019 (EXTBOB) : Faceplate selection for configuration of 
   // analog signal atleast one selected newly added
   IF (NOT #FP_SEL.X3 OR #FP_SEL.Type2) AND NOT #FP_SEL.X1 AND NOT #FP_SEL.X2 THEN
       #FP_SEL.X1 := TRUE;
   END_IF;
END_REGION

REGION Network 14: Check Signal X1 <-> X3
   // ENO of a box is taken as its EN; it also drops when the box reports an error
   #DummyReal_1 := #X1 - #X3;
   #DummyReal_2 := ABS(#DummyReal_1);
END_REGION

REGION Network 15: Delay Time X1<->X3 Alarm
   // Ignor if type-2 Sensor Selecetd
   // 
   // Build 002 - 17. Jun 2019 (EXTBOB) : Faceplate selection & Signal enable 
   // flag added
   "ACESYS_SecTimer_INT"(START := (#DummyReal_2 > #FP_PARM.MaxDiff) AND #FP_SEL.Type3 AND #FP_SEL.X1 AND #FP_SEL.X3 AND #X1_OK AND #X3_OK,
                         SEC := #Sec_Pulse,
                         PRE := #FP_PARM.AL_Delay_Pre,
                         Mem := #Sig1_3_TimerMEM,
                         ACC => #FP_PARM.AL_Delay_Acc,
                         DN => #Sig1_3_NotOK,
                         TT => #DummyBool);
END_REGION

REGION Network 16: Check Signal X1 <-> X2
   // ENO of a box is taken as its EN; it also drops when the box reports an error
   #DummyReal_1 := #X1 - #X2;
   #DummyReal_2 := ABS(#DummyReal_1);
END_REGION

REGION Network 17: Delay Time X1<->X2 Alarm
   // Build 002 - 17. Jun 2019 (EXTBOB) : Faceplate selection & Signal enable 
   // flag added
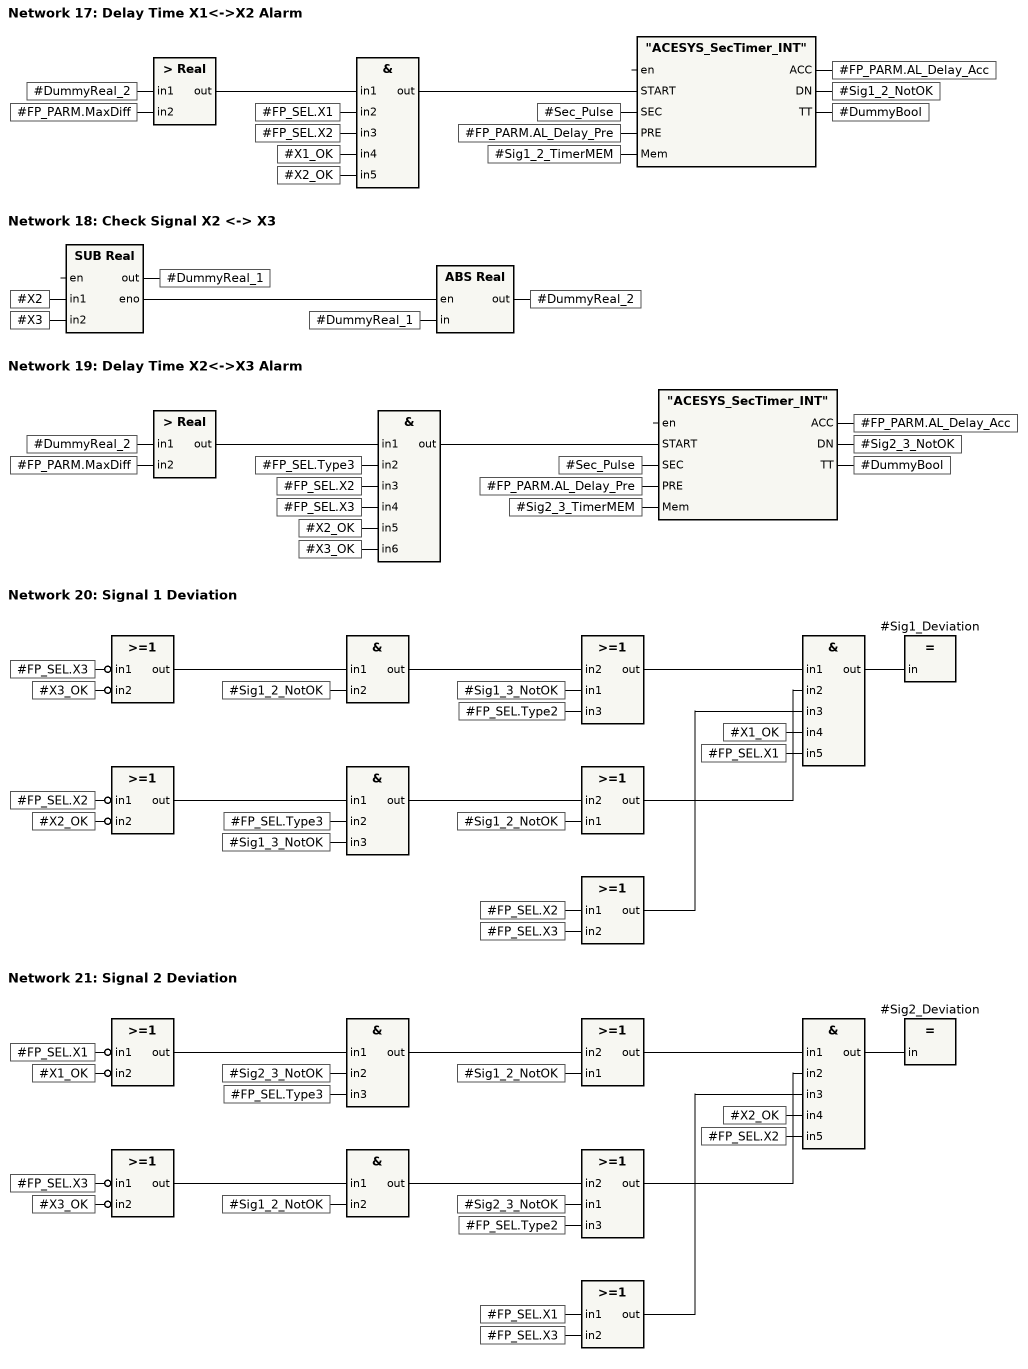
   "ACESYS_SecTimer_INT"(START := (#DummyReal_2 > #FP_PARM.MaxDiff) AND #FP_SEL.X1 AND #FP_SEL.X2 AND #X1_OK AND #X2_OK,
                         SEC := #Sec_Pulse,
                         PRE := #FP_PARM.AL_Delay_Pre,
                         Mem := #Sig1_2_TimerMEM,
                         ACC => #FP_PARM.AL_Delay_Acc,
                         DN => #Sig1_2_NotOK,
                         TT => #DummyBool);
END_REGION

REGION Network 18: Check Signal X2 <-> X3
   // ENO of a box is taken as its EN; it also drops when the box reports an error
   #DummyReal_1 := #X2 - #X3;
   #DummyReal_2 := ABS(#DummyReal_1);
END_REGION

REGION Network 19: Delay Time X2<->X3 Alarm
   // Ignor if type-2 Sensor Selecetd
   // 
   // Build 002 - 17. Jun 2019 (EXTBOB) : Faceplate selection & Signal enable 
   // flag added
   "ACESYS_SecTimer_INT"(START := (#DummyReal_2 > #FP_PARM.MaxDiff) AND #FP_SEL.Type3 AND #FP_SEL.X2 AND #FP_SEL.X3 AND #X2_OK AND #X3_OK,
                         SEC := #Sec_Pulse,
                         PRE := #FP_PARM.AL_Delay_Pre,
                         Mem := #Sig2_3_TimerMEM,
                         ACC => #FP_PARM.AL_Delay_Acc,
                         DN => #Sig2_3_NotOK,
                         TT => #DummyBool);
END_REGION

REGION Network 20: Signal 1 Deviation
   // Build 002 - 17. Jun 2019 (EXTBOB) : Faceplate selection & Signal enable 
   // flag added
   #Sig1_Deviation := (((NOT #FP_SEL.X3 OR NOT #X3_OK) AND #Sig1_2_NotOK) OR #Sig1_3_NotOK OR #FP_SEL.Type2) AND (((NOT #FP_SEL.X2 OR NOT #X2_OK) AND #FP_SEL.Type3 AND #Sig1_3_NotOK) OR #Sig1_2_NotOK) AND (#FP_SEL.X2 OR #FP_SEL.X3) AND #X1_OK AND #FP_SEL.X1;
END_REGION

REGION Network 21: Signal 2 Deviation
   // Build 002 - 17. Jun 2019 (EXTBOB) : Faceplate selection & Signal enable flag 
   // added
   #Sig2_Deviation := (((NOT #FP_SEL.X1 OR NOT #X1_OK) AND #Sig2_3_NotOK AND #FP_SEL.Type3) OR #Sig1_2_NotOK) AND (((NOT #FP_SEL.X3 OR NOT #X3_OK) AND #Sig1_2_NotOK) OR #Sig2_3_NotOK OR #FP_SEL.Type2) AND (#FP_SEL.X1 OR #FP_SEL.X3) AND #X2_OK AND #FP_SEL.X2;
END_REGION

REGION Network 22: Signal 3 Deviation
   // Build 002 - 17. Jun 2019 (EXTBOB) : Faceplate selection & Signal enable flag 
   // added
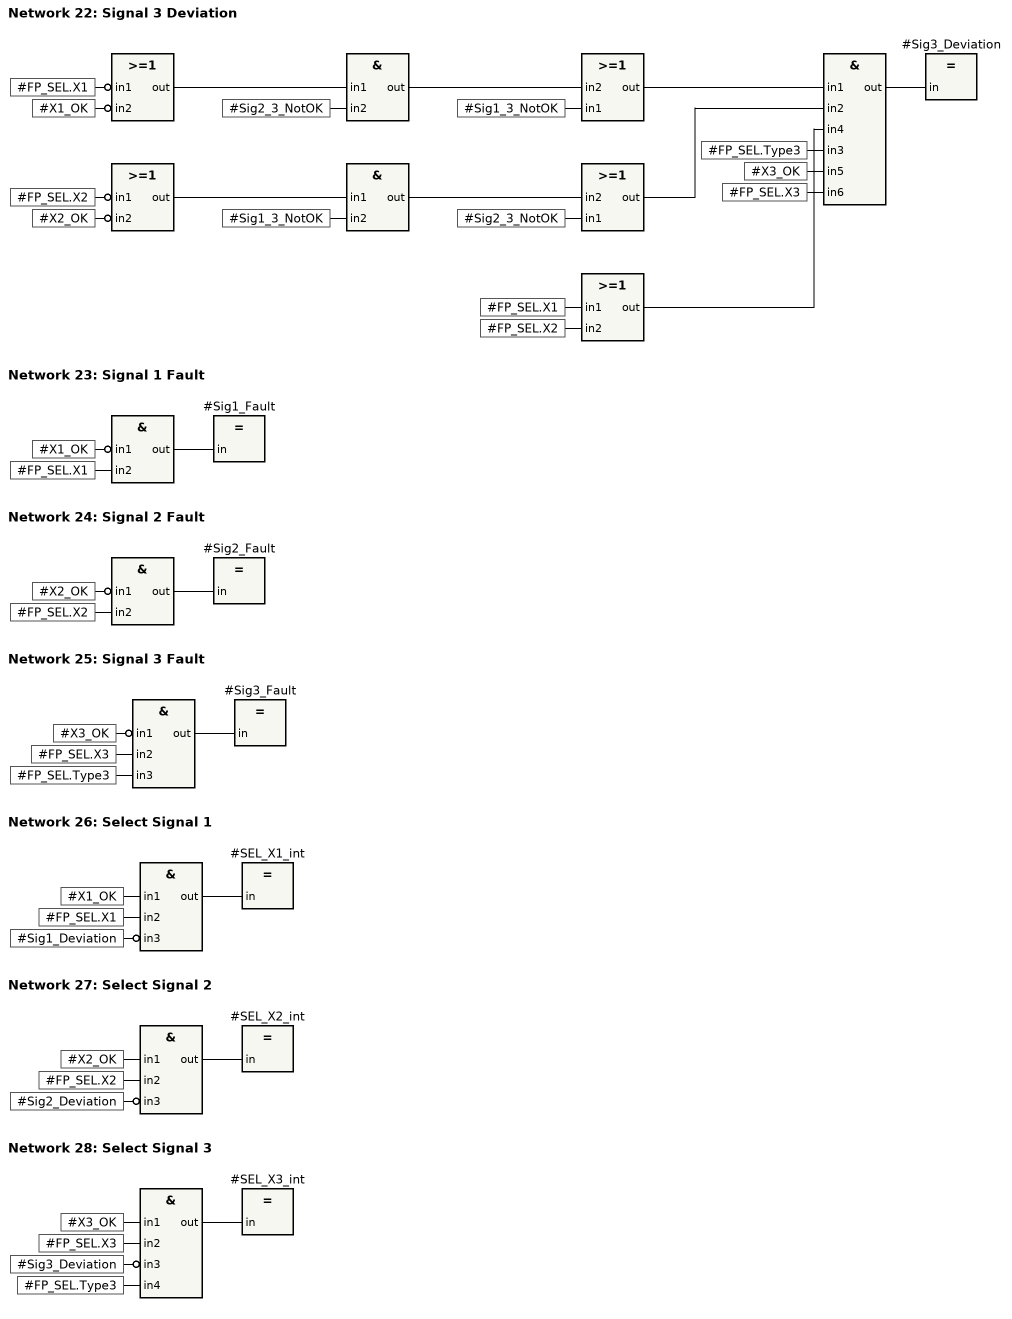
   #Sig3_Deviation := (((NOT #FP_SEL.X1 OR NOT #X1_OK) AND #Sig2_3_NotOK) OR #Sig1_3_NotOK) AND (((NOT #FP_SEL.X2 OR NOT #X2_OK) AND #Sig1_3_NotOK) OR #Sig2_3_NotOK) AND (#FP_SEL.X1 OR #FP_SEL.X2) AND #FP_SEL.Type3 AND #X3_OK AND #FP_SEL.X3;
END_REGION

REGION Network 23: Signal 1 Fault
   // Build 002 - 17. Jun 2019 (EXTBOB) : Signal-1 fault flag newly added
   #Sig1_Fault := NOT #X1_OK AND #FP_SEL.X1;
END_REGION

REGION Network 24: Signal 2 Fault
   // Build 002 - 17. Jun 2019 (EXTBOB) : Signal-2 fault flag newly added
   #Sig2_Fault := NOT #X2_OK AND #FP_SEL.X2;
END_REGION

REGION Network 25: Signal 3 Fault
   // Build 002 - 17. Jun 2019 (EXTBOB) : Signal-3 fault flag newly added
   #Sig3_Fault := NOT #X3_OK AND #FP_SEL.X3 AND #FP_SEL.Type3;
END_REGION

REGION Network 26: Select Signal 1
   #SEL_X1_int := #X1_OK AND #FP_SEL.X1 AND NOT #Sig1_Deviation;
END_REGION

REGION Network 27: Select Signal 2
   #SEL_X2_int := #X2_OK AND #FP_SEL.X2 AND NOT #Sig2_Deviation;
END_REGION

REGION Network 28: Select Signal 3
   #SEL_X3_int := #X3_OK AND #FP_SEL.X3 AND NOT #Sig3_Deviation AND #FP_SEL.Type3;
END_REGION

REGION Network 29: Clear Values
   // *****Calculate Average*****
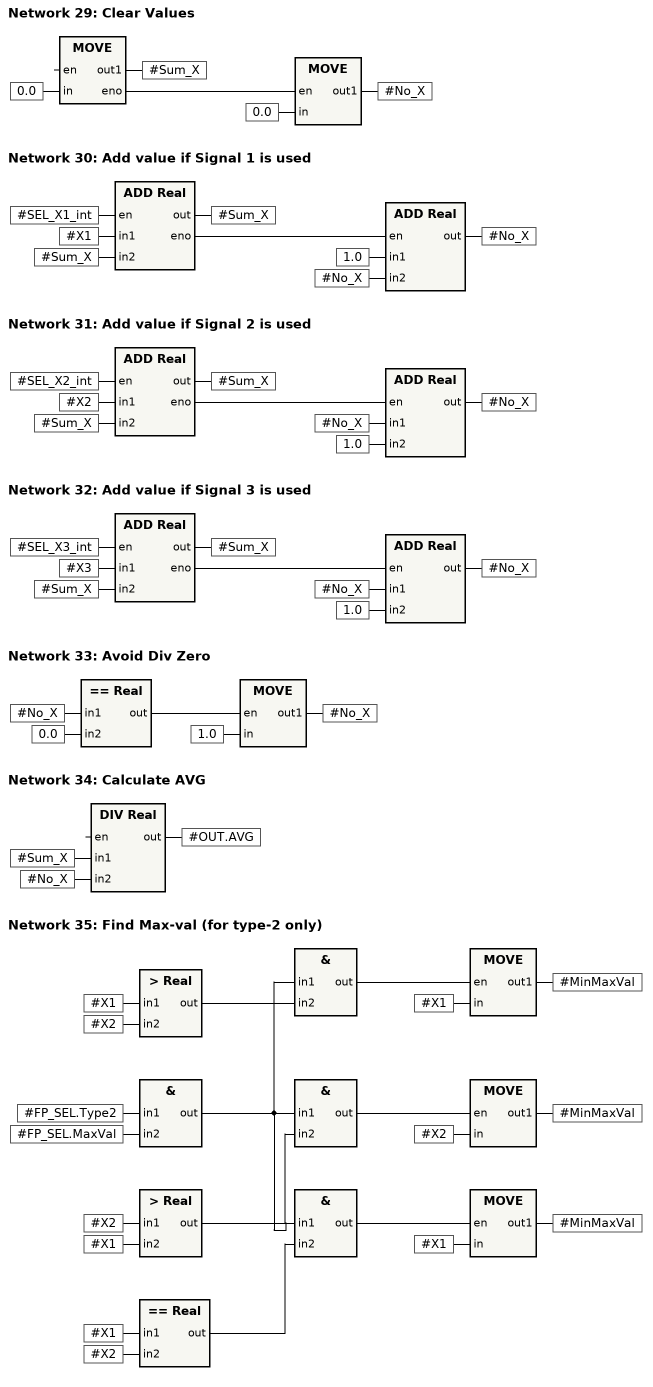
   // ENO of a box is taken as its EN; it also drops when the box reports an error
   #Sum_X := 0.0;
   #No_X := 0.0;
END_REGION

REGION Network 30: Add value if Signal 1 is used
   // ENO of a box is taken as its EN; it also drops when the box reports an error
   IF #SEL_X1_int THEN
       #Sum_X := #X1 + #Sum_X;
       #No_X := 1.0 + #No_X;
   END_IF;
END_REGION

REGION Network 31: Add value if Signal 2 is used
   // ENO of a box is taken as its EN; it also drops when the box reports an error
   IF #SEL_X2_int THEN
       #Sum_X := #X2 + #Sum_X;
       #No_X := #No_X + 1.0;
   END_IF;
END_REGION

REGION Network 32: Add value if Signal 3 is used
   // ENO of a box is taken as its EN; it also drops when the box reports an error
   IF #SEL_X3_int THEN
       #Sum_X := #X3 + #Sum_X;
       #No_X := #No_X + 1.0;
   END_IF;
END_REGION

REGION Network 33: Avoid Div Zero
   IF #No_X = 0.0 THEN #No_X := 1.0; END_IF;
END_REGION

REGION Network 34: Calculate AVG
   #OUT.AVG := #Sum_X / #No_X;
END_REGION

REGION Network 35: Find Max-val (for type-2 only)
   #_w1 := #FP_SEL.Type2 AND #FP_SEL.MaxVal;
   IF #_w1 AND (#X1 > #X2) THEN #MinMaxVal := #X1; END_IF;
   IF #_w1 AND (#X2 > #X1) THEN #MinMaxVal := #X2; END_IF;
   IF #_w1 AND (#X1 = #X2) THEN #MinMaxVal := #X1; END_IF;
END_REGION

REGION Network 36: Find Min-val (for type-2 only)
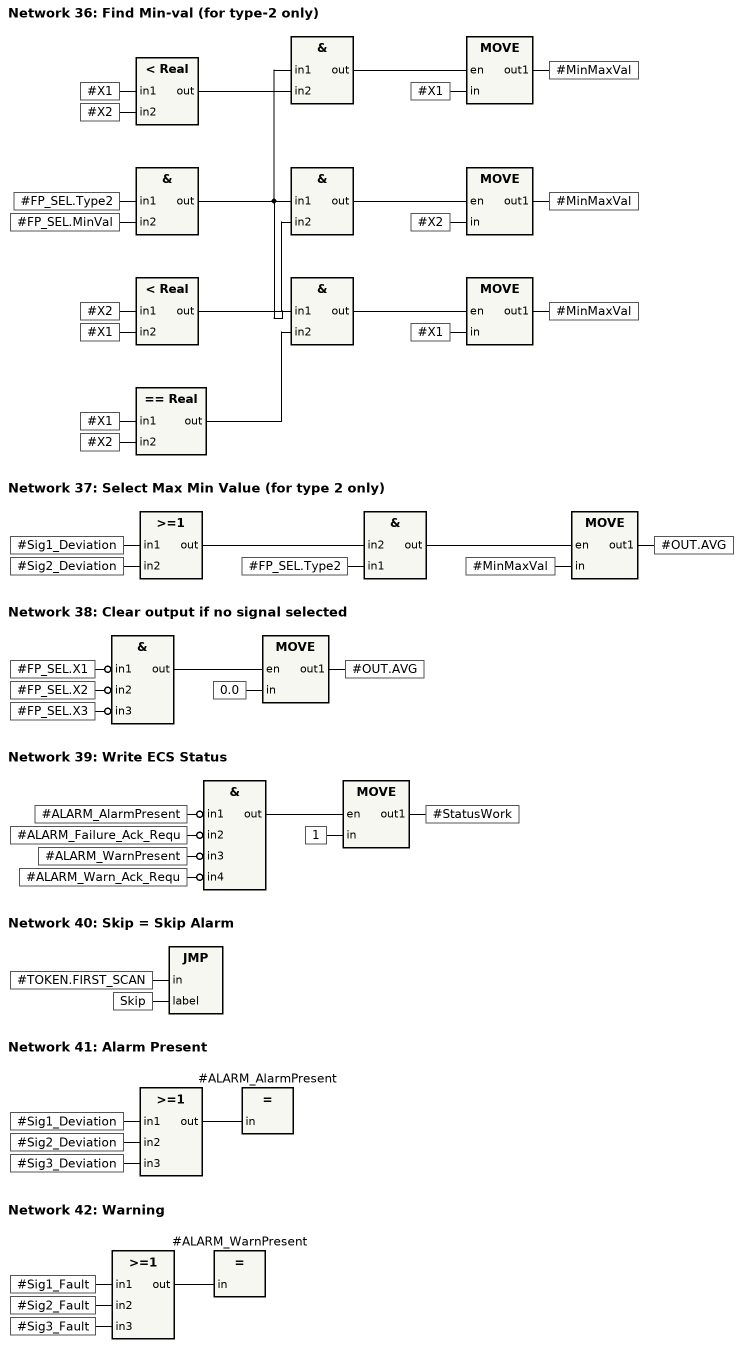
   #_w1 := #FP_SEL.Type2 AND #FP_SEL.MinVal;
   IF #_w1 AND (#X1 < #X2) THEN #MinMaxVal := #X1; END_IF;
   IF #_w1 AND (#X2 < #X1) THEN #MinMaxVal := #X2; END_IF;
   IF #_w1 AND (#X1 = #X2) THEN #MinMaxVal := #X1; END_IF;
END_REGION

REGION Network 37: Select Max Min Value (for type 2 only)
   IF (#Sig1_Deviation OR #Sig2_Deviation) AND #FP_SEL.Type2 THEN #OUT.AVG := #MinMaxVal; END_IF;
END_REGION

REGION Network 38: Clear output if no signal selected
   IF NOT #FP_SEL.X1 AND NOT #FP_SEL.X2 AND NOT #FP_SEL.X3 THEN #OUT.AVG := 0.0; END_IF;
END_REGION

REGION Network 39: Write ECS Status
   // Build 002 - 17. Jun 2019 (EXTBOB) : Negate of Alarm warning Present and Alarm 
   // Warning Ack required added
   IF NOT #ALARM_AlarmPresent AND NOT #ALARM_Failure_Ack_Requ AND NOT #ALARM_WarnPresent AND NOT #ALARM_Warn_Ack_Requ THEN
       #StatusWork := 1;
   END_IF;
END_REGION

REGION Network 40: Skip = Skip Alarm
   IF #TOKEN.FIRST_SCAN THEN GOTO Skip; END_IF;
END_REGION

REGION Network 41: Alarm Present
   #ALARM_AlarmPresent := #Sig1_Deviation OR #Sig2_Deviation OR #Sig3_Deviation;
END_REGION

REGION Network 42: Warning
   // Build 002 - 17. Jun 2019 (EXTBOB) : Signal-1 fault warning newly added
   #ALARM_WarnPresent := #Sig1_Fault OR #Sig2_Fault OR #Sig3_Fault;
END_REGION

REGION Network 43: Skip = Skip Alarm
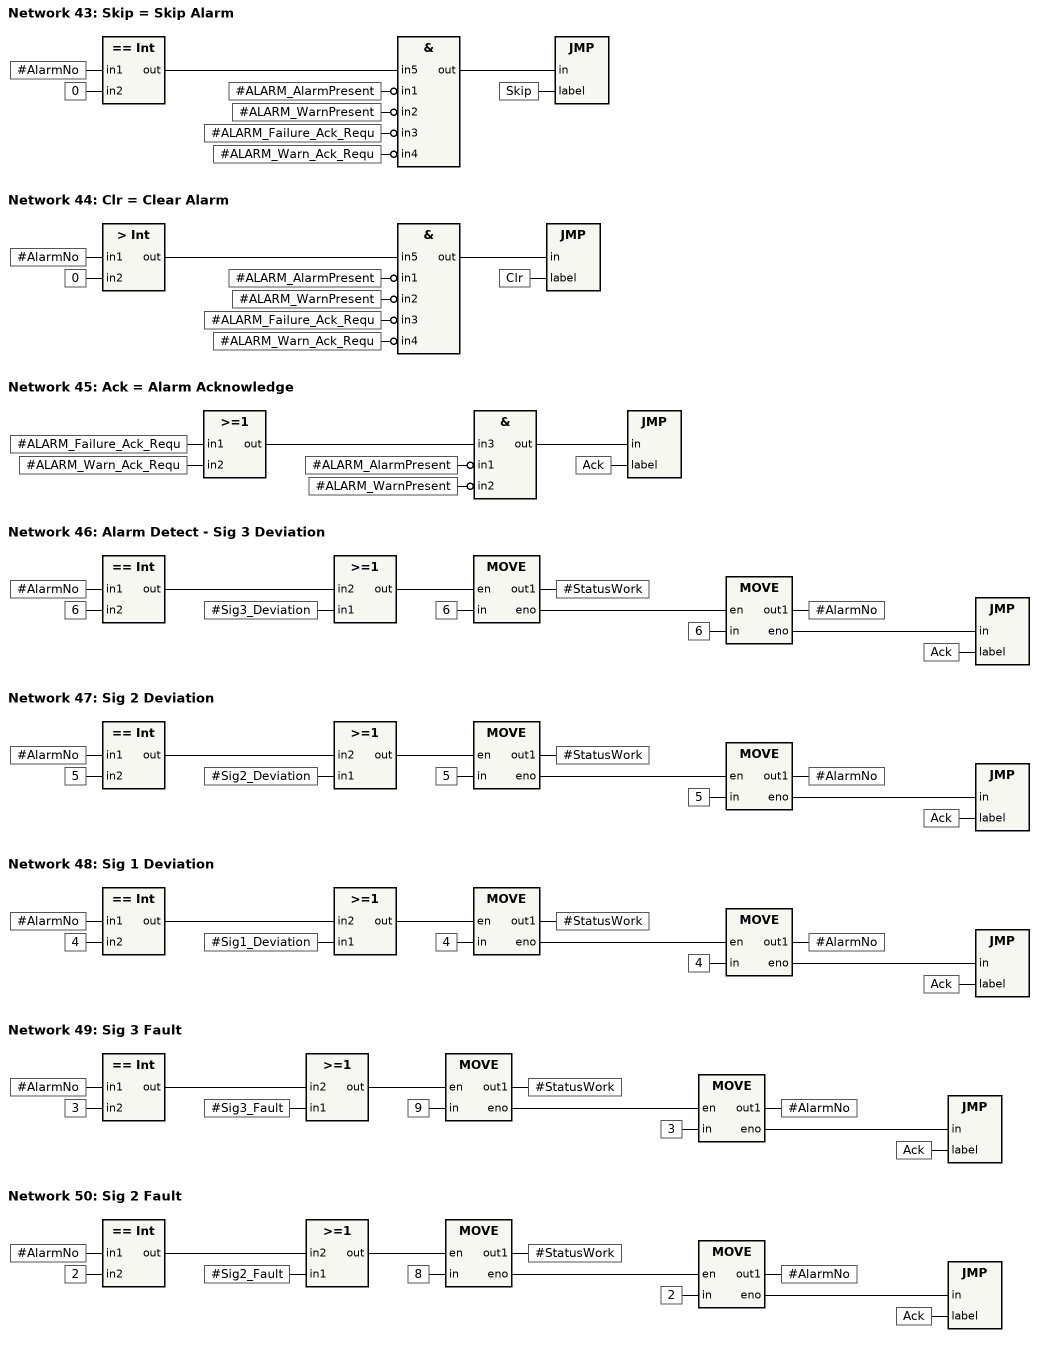
   IF (#AlarmNo = 0) AND NOT #ALARM_AlarmPresent AND NOT #ALARM_WarnPresent AND NOT #ALARM_Failure_Ack_Requ AND NOT #ALARM_Warn_Ack_Requ THEN
       GOTO Skip;
   END_IF;
END_REGION

REGION Network 44: Clr = Clear Alarm
   IF (#AlarmNo > 0) AND NOT #ALARM_AlarmPresent AND NOT #ALARM_WarnPresent AND NOT #ALARM_Failure_Ack_Requ AND NOT #ALARM_Warn_Ack_Requ THEN
       GOTO Clr;
   END_IF;
END_REGION

REGION Network 45: Ack = Alarm Acknowledge
   IF (#ALARM_Failure_Ack_Requ OR #ALARM_Warn_Ack_Requ) AND NOT #ALARM_AlarmPresent AND NOT #ALARM_WarnPresent THEN
       GOTO Ack;
   END_IF;
END_REGION

REGION Network 46: Alarm Detect - Sig 3 Deviation
   // ENO of a box is taken as its EN; it also drops when the box reports an error
   #_w1 := (#AlarmNo = 6) OR #Sig3_Deviation;
   IF #_w1 THEN
       #StatusWork := 6;
       #AlarmNo := 6;
       GOTO Ack;
   END_IF;
END_REGION

REGION Network 47: Sig 2 Deviation
   // ENO of a box is taken as its EN; it also drops when the box reports an error
   #_w1 := (#AlarmNo = 5) OR #Sig2_Deviation;
   IF #_w1 THEN
       #StatusWork := 5;
       #AlarmNo := 5;
       GOTO Ack;
   END_IF;
END_REGION

REGION Network 48: Sig 1 Deviation
   // ENO of a box is taken as its EN; it also drops when the box reports an error
   #_w1 := (#AlarmNo = 4) OR #Sig1_Deviation;
   IF #_w1 THEN
       #StatusWork := 4;
       #AlarmNo := 4;
       GOTO Ack;
   END_IF;
END_REGION

REGION Network 49: Sig 3 Fault
   // Build 002 - 17. Jun 2019 (EXTBOB) : Signal-3 fault alarm detect newly added
   // ENO of a box is taken as its EN; it also drops when the box reports an error
   #_w1 := (#AlarmNo = 3) OR #Sig3_Fault;
   IF #_w1 THEN
       #StatusWork := 9;
       #AlarmNo := 3;
       GOTO Ack;
   END_IF;
END_REGION

REGION Network 50: Sig 2 Fault
   // Build 002 - 17. Jun 2019 (EXTBOB) : Signal-2 fault alarm detect newly added
   // ENO of a box is taken as its EN; it also drops when the box reports an error
   #_w1 := (#AlarmNo = 2) OR #Sig2_Fault;
   IF #_w1 THEN
       #StatusWork := 8;
       #AlarmNo := 2;
       GOTO Ack;
   END_IF;
END_REGION

REGION Network 51: Sig 1 Fault
   // Build 002 - 17. Jun 2019 (EXTBOB) : Signal-1 fault alarm detect newly added
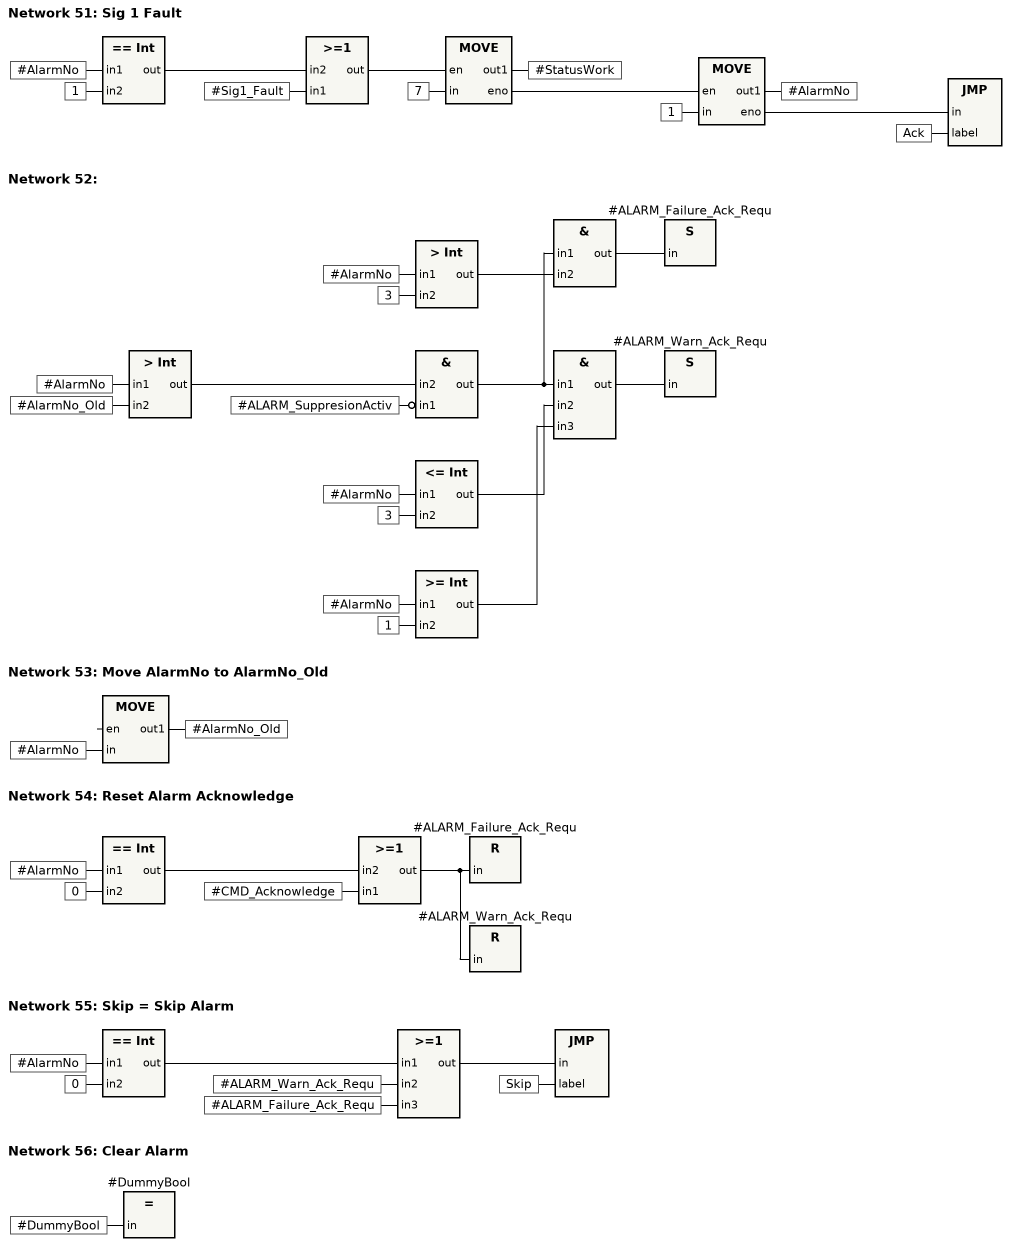
   // ENO of a box is taken as its EN; it also drops when the box reports an error
   #_w1 := (#AlarmNo = 1) OR #Sig1_Fault;
   IF #_w1 THEN
       #StatusWork := 7;
       #AlarmNo := 1;
       GOTO Ack;
   END_IF;
END_REGION

REGION Network 52
   // >>>>>Alarm Acknowledge<<<<<
   // 
   // Build 002 - 17. Jun 2019 (EXTBOB) : Alarm Warning Acknowlege Required updated
   Ack:
   #_w1 := (#AlarmNo > #AlarmNo_Old) AND NOT #ALARM_SuppresionActiv;
   IF #_w1 AND (#AlarmNo > 3) THEN #ALARM_Failure_Ack_Requ := TRUE; END_IF;
   IF #_w1 AND (#AlarmNo <= 3) AND (#AlarmNo >= 1) THEN #ALARM_Warn_Ack_Requ := TRUE; END_IF;
END_REGION

REGION Network 53: Move AlarmNo to AlarmNo_Old
   #AlarmNo_Old := #AlarmNo;
END_REGION

REGION Network 54: Reset Alarm Acknowledge
   IF (#AlarmNo = 0) OR #CMD_Acknowledge THEN
       #ALARM_Failure_Ack_Requ := FALSE;
       #ALARM_Warn_Ack_Requ := FALSE;
   END_IF;
END_REGION

REGION Network 55: Skip = Skip Alarm
   IF (#AlarmNo = 0) OR #ALARM_Warn_Ack_Requ OR #ALARM_Failure_Ack_Requ THEN GOTO Skip; END_IF;
END_REGION

REGION Network 56: Clear Alarm
   Clr:
   #DummyBool := #DummyBool;
END_REGION

REGION Network 57
   // Build 002 - 17. Jun 2019 (EXTBOB) : Signal fault 1,2,3 also added to clear the 
   // alarm number
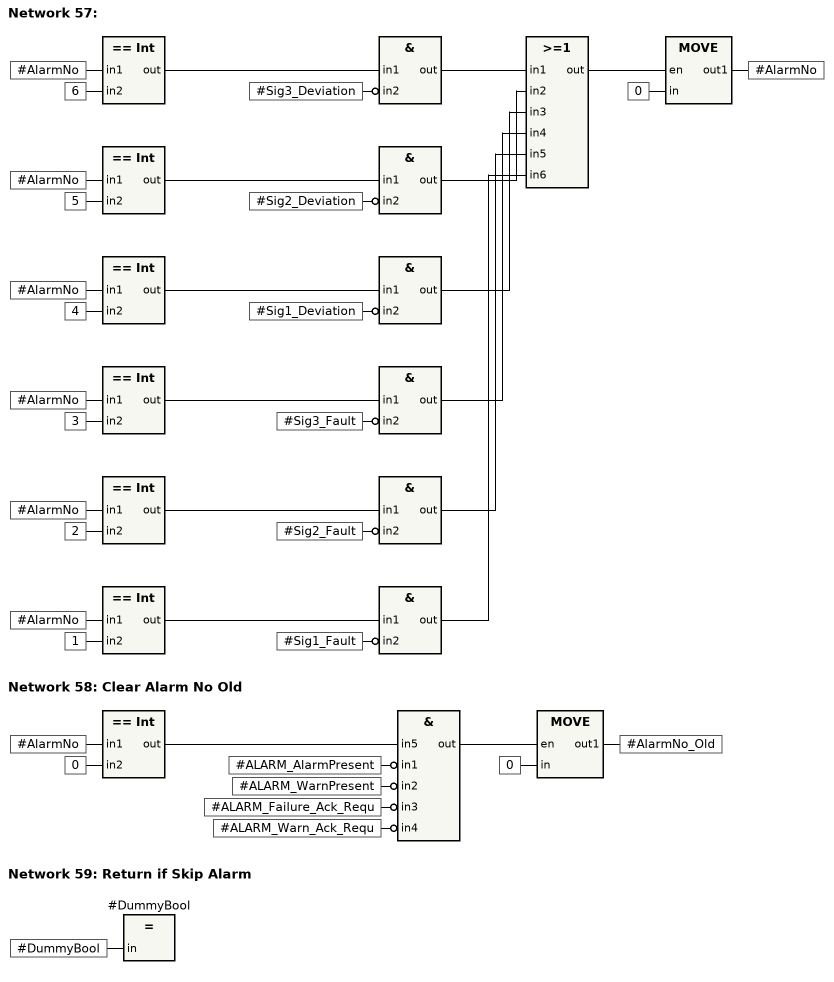
   IF ((#AlarmNo = 6) AND NOT #Sig3_Deviation) OR ((#AlarmNo = 5) AND NOT #Sig2_Deviation) OR ((#AlarmNo = 4) AND NOT #Sig1_Deviation) OR ((#AlarmNo = 3) AND NOT #Sig3_Fault) OR ((#AlarmNo = 2) AND NOT #Sig2_Fault) OR ((#AlarmNo = 1) AND NOT #Sig1_Fault) THEN
       #AlarmNo := 0;
   END_IF;
END_REGION

REGION Network 58: Clear Alarm No Old
   IF (#AlarmNo = 0) AND NOT #ALARM_AlarmPresent AND NOT #ALARM_WarnPresent AND NOT #ALARM_Failure_Ack_Requ AND NOT #ALARM_Warn_Ack_Requ THEN
       #AlarmNo_Old := 0;
   END_IF;
END_REGION

REGION Network 59: Return if Skip Alarm
   Skip:
   #DummyBool := #DummyBool;
END_REGION

REGION Network 60: Alarm Output
   // Set Output Signals
   // 
   // Build 002 - 17. Jun 2019 (EXTBOB) : Signal Fault 1,2,3 also added to reset the 
   // output
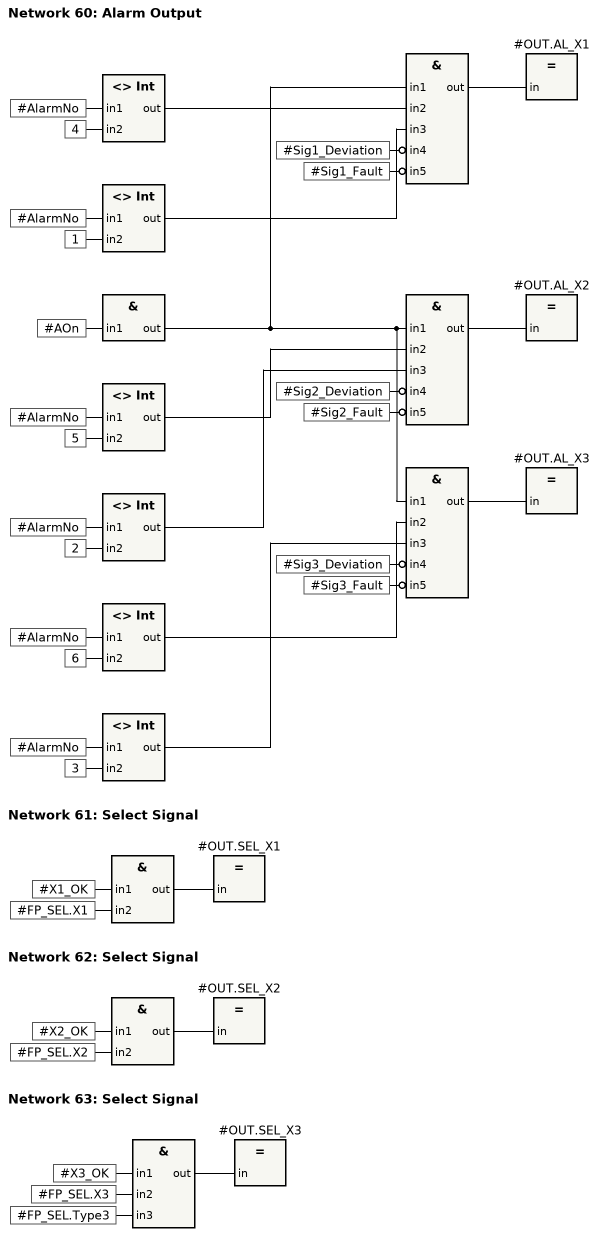
   #OUT.AL_X1 := #AOn AND (#AlarmNo <> 4) AND (#AlarmNo <> 1) AND NOT #Sig1_Deviation AND NOT #Sig1_Fault;
   #OUT.AL_X2 := #AOn AND (#AlarmNo <> 5) AND (#AlarmNo <> 2) AND NOT #Sig2_Deviation AND NOT #Sig2_Fault;
   #OUT.AL_X3 := #AOn AND (#AlarmNo <> 6) AND (#AlarmNo <> 3) AND NOT #Sig3_Deviation AND NOT #Sig3_Fault;
END_REGION

REGION Network 61: Select Signal
   #OUT.SEL_X1 := #X1_OK AND #FP_SEL.X1;
END_REGION

REGION Network 62: Select Signal
   #OUT.SEL_X2 := #X2_OK AND #FP_SEL.X2;
END_REGION

REGION Network 63: Select Signal
   #OUT.SEL_X3 := #X3_OK AND #FP_SEL.X3 AND #FP_SEL.Type3;
END_REGION

REGION Network 64: Update Boolean Data in MSW - Bit 16-19: Mode
   // 0 = Auto
   // 1 = Single Start
   // 2 = Manual
   // 3 = Local
   // 4 = Test Mode
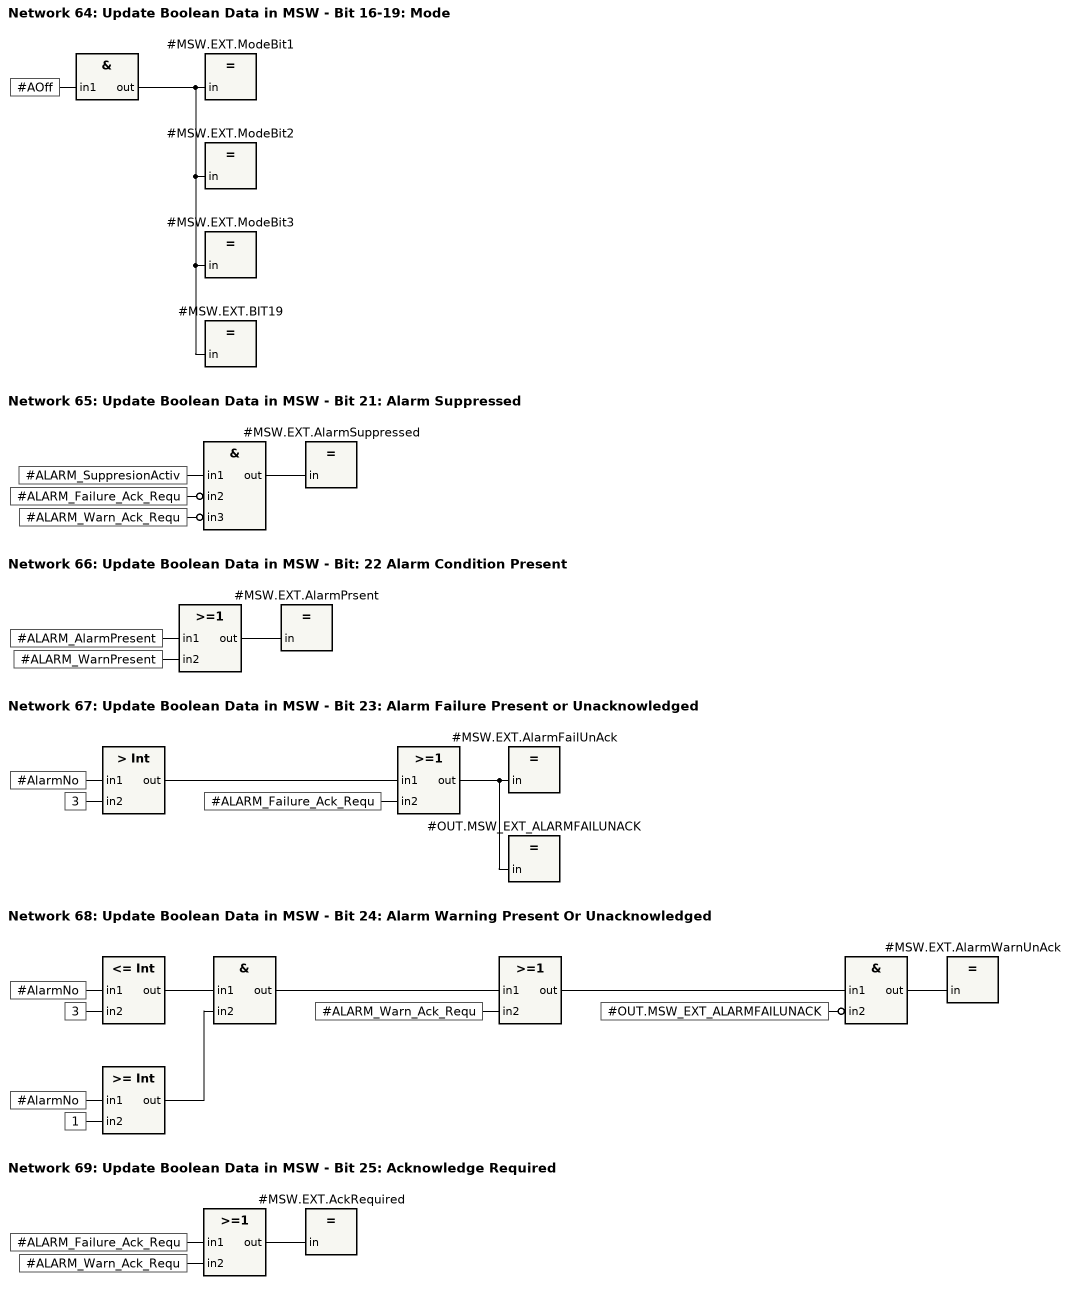
   #MSW.EXT.ModeBit1 := #AOff;
   #MSW.EXT.ModeBit2 := #AOff;
   #MSW.EXT.ModeBit3 := #AOff;
   #MSW.EXT.BIT19 := #AOff;
END_REGION

REGION Network 65: Update Boolean Data in MSW - Bit 21: Alarm Suppressed
   #MSW.EXT.AlarmSuppressed := #ALARM_SuppresionActiv AND NOT #ALARM_Failure_Ack_Requ AND NOT #ALARM_Warn_Ack_Requ;
END_REGION

REGION Network 66: Update Boolean Data in MSW - Bit: 22 Alarm Condition Present
   #MSW.EXT.AlarmPrsent := #ALARM_AlarmPresent OR #ALARM_WarnPresent;
END_REGION

REGION Network 67: Update Boolean Data in MSW - Bit 23: Alarm Failure Present or Unacknowledged
   #MSW.EXT.AlarmFailUnAck := (#AlarmNo > 3) OR #ALARM_Failure_Ack_Requ;
   #OUT.MSW_EXT_ALARMFAILUNACK := #MSW.EXT.AlarmFailUnAck;
END_REGION

REGION Network 68: Update Boolean Data in MSW - Bit 24: Alarm Warning Present Or Unacknowledged
   // Build 002 - 17. Jun 2019 (EXTBOB) : Alarm Warning UnAcknowlege updated with Alarm No 1,2,3
   #MSW.EXT.AlarmWarnUnAck := (((#AlarmNo <= 3) AND (#AlarmNo >= 1)) OR #ALARM_Warn_Ack_Requ) AND NOT #OUT.MSW_EXT_ALARMFAILUNACK;
END_REGION

REGION Network 69: Update Boolean Data in MSW - Bit 25: Acknowledge Required
   #MSW.EXT.AckRequired := #ALARM_Failure_Ack_Requ OR #ALARM_Warn_Ack_Requ;
END_REGION

REGION Network 70: Update Boolean Data in MSW - Bit 26,27: Maintenence/Operation
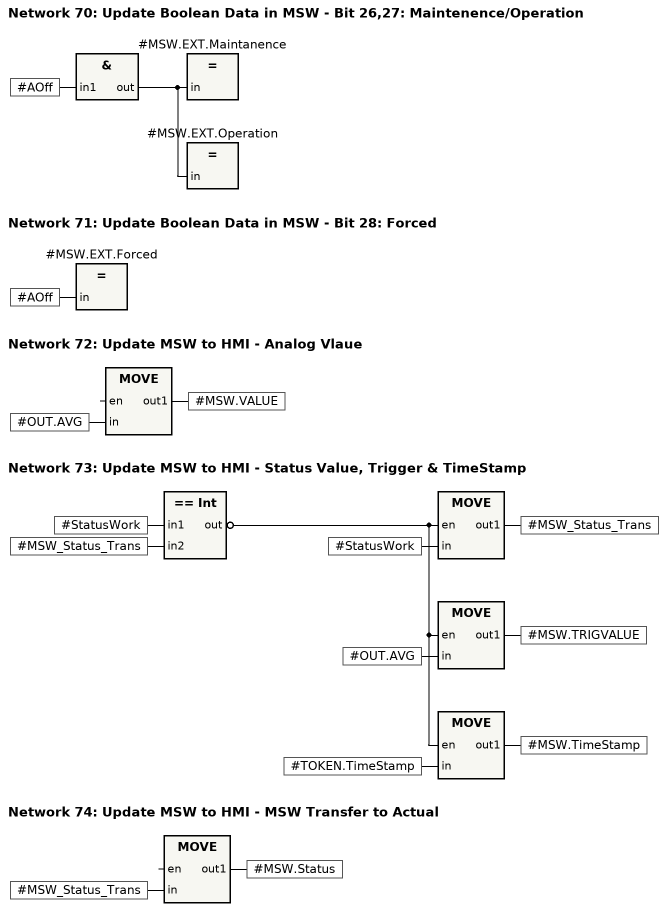
   #MSW.EXT.Maintanence := #AOff;
   #MSW.EXT.Operation := #AOff;
END_REGION

REGION Network 71: Update Boolean Data in MSW - Bit 28: Forced
   #MSW.EXT.Forced := #AOff;
END_REGION

REGION Network 72: Update MSW to HMI - Analog Vlaue
   #MSW.VALUE := #OUT.AVG;
END_REGION

REGION Network 73: Update MSW to HMI - Status Value, Trigger & TimeStamp
   #_w1 := NOT (#StatusWork = #MSW_Status_Trans);
   IF #_w1 THEN
       #MSW_Status_Trans := #StatusWork;
       #MSW.TRIGVALUE := #OUT.AVG;
       #MSW.TimeStamp := #TOKEN.TimeStamp;
   END_IF;
END_REGION

REGION Network 74: Update MSW to HMI - MSW Transfer to Actual
   #MSW.Status := #MSW_Status_Trans;
END_REGION

REGION Network 75: Write Stat to OUT
